   DATA[467,23] := 980.5178;
   DATA[467,24] := 2.0;
   DATA[467,25] := 2.0;
   DATA[467,26] := 7.878621;
   DATA[467,27] := 145.091;
   DATA[467,28] := 263.5222;
   DATA[467,29] := 12.11228;
   DATA[467,30] := 1.729557;
   DATA[467,31] := 1.292046;
   DATA[467,32] := 0.7353967;
   DATA[467,33] := 0.3065048;
   DATA[467,34] := 2.0;
   DATA[467,35] := 251.2817;
   DATA[467,36] := 1.746067;
   DATA[467,37] := 190.0634;
   DATA[467,38] := 0.000128152;
   DATA[467,39] := 1.0;
   DATA[468,0] := 2.44243;
   DATA[468,1] := 530.9328;
   DATA[468,2] := 2.0;
   DATA[468,3] := 2.0;
   DATA[468,4] := 262.1764;
   DATA[468,5] := 8.394835;
   DATA[468,6] := 327.9928;
   DATA[468,7] := 2.440521;
   DATA[468,8] := 2.0;
   DATA[468,9] := 2.0;
   DATA[468,10] := 2.0;
   DATA[468,11] := 19.69396;
   DATA[468,12] := 2.213881;
   DATA[468,13] := 980.0773;
   DATA[468,14] := 1.0;
   DATA[468,15] := 2.0;
   DATA[468,16] := 1.0;
   DATA[468,17] := 1.0;
   DATA[468,18] := 1.0;
   DATA[468,19] := 2.0;
   DATA[468,20] := 148.808;
   DATA[468,21] := 155.96;
   DATA[468,22] := 1.720565;
   DATA[468,23] := 980.5563;
   DATA[468,24] := 2.0;
   DATA[468,25] := 2.0;
   DATA[468,26] := 7.878621;
   DATA[468,27] := 145.091;
   DATA[468,28] := 263.5222;
   DATA[468,29] := 12.11228;
   DATA[468,30] := 1.730838;
   DATA[468,31] := 1.293198;
   DATA[468,32] := 0.7353967;
   DATA[468,33] := 0.3065048;
   DATA[468,34] := 2.0;
   DATA[468,35] := 251.2817;
   DATA[468,36] := 1.826162;
   DATA[468,37] := 190.0634;
   DATA[468,38] := 0.000128152;
   DATA[468,39] := 1.0;
   DATA[469,0] := 2.427377;
   DATA[469,1] := 530.3832;
   DATA[469,2] := 2.0;
   DATA[469,3] := 2.0;
   DATA[469,4] := 262.1764;
   DATA[469,5] := 8.394835;
   DATA[469,6] := 327.9928;
   DATA[469,7] := 2.440137;
   DATA[469,8] := 2.0;
   DATA[469,9] := 2.0;
   DATA[469,10] := 2.0;
   DATA[469,11] := 19.69396;
   DATA[469,12] := 2.213881;
   DATA[469,13] := 979.9971;
   DATA[469,14] := 1.0;
   DATA[469,15] := 2.0;
   DATA[469,16] := 1.0;
   DATA[469,17] := 1.0;
   DATA[469,18] := 1.0;
   DATA[469,19] := 2.0;
   DATA[469,20] := 148.808;
   DATA[469,21] := 155.96;
   DATA[469,22] := 1.720565;
   DATA[469,23] := 980.5563;
   DATA[469,24] := 2.0;
   DATA[469,25] := 2.0;
   DATA[469,26] := 7.878621;
   DATA[469,27] := 145.091;
   DATA[469,28] := 263.5222;
   DATA[469,29] := 12.11228;
   DATA[469,30] := 1.730838;
   DATA[469,31] := 1.296657;
   DATA[469,32] := 0.7353967;
   DATA[469,33] := 0.3065048;
   DATA[469,34] := 2.0;
   DATA[469,35] := 251.2817;
   DATA[469,36] := 1.826162;
   DATA[469,37] := 190.0634;
   DATA[469,38] := 0.000128152;
   DATA[469,39] := 1.0;
   DATA[470,0] := 2.427377;
   DATA[470,1] := 530.6188;
   DATA[470,2] := 2.0;
   DATA[470,3] := 2.0;
   DATA[470,4] := 262.1764;
   DATA[470,5] := 8.394835;
   DATA[470,6] := 327.9928;
   DATA[470,7] := 2.440137;
   DATA[470,8] := 2.0;
   DATA[470,9] := 2.0;
   DATA[470,10] := 2.0;
   DATA[470,11] := 19.65235;
   DATA[470,12] := 2.213881;
   DATA[470,13] := 979.9571;
   DATA[470,14] := 1.0;
   DATA[470,15] := 2.0;
   DATA[470,16] := 1.0;
   DATA[470,17] := 1.0;
   DATA[470,18] := 1.0;
   DATA[470,19] := 2.0;
   DATA[470,20] := 148.808;
   DATA[470,21] := 155.96;
   DATA[470,22] := 1.720565;
   DATA[470,23] := 980.364;
   DATA[470,24] := 2.0;
   DATA[470,25] := 2.0;
   DATA[470,26] := 7.878621;
   DATA[470,27] := 145.091;
   DATA[470,28] := 263.5222;
   DATA[470,29] := 12.11228;
   DATA[470,30] := 1.730838;
   DATA[470,31] := 1.289868;
   DATA[470,32] := 0.7353967;
   DATA[470,33] := 0.3065048;
   DATA[470,34] := 2.0;
   DATA[470,35] := 251.2817;
   DATA[470,36] := 1.762086;
   DATA[470,37] := 190.0634;
   DATA[470,38] := 0.000128152;
   DATA[470,39] := 1.0;
   DATA[471,0] := 2.427377;
   DATA[471,1] := 530.3047;
   DATA[471,2] := 2.0;
   DATA[471,3] := 2.0;
   DATA[471,4] := 262.1764;
   DATA[471,5] := 8.394835;
   DATA[471,6] := 327.9928;
   DATA[471,7] := 2.440137;
   DATA[471,8] := 2.0;
   DATA[471,9] := 2.0;
   DATA[471,10] := 2.0;
   DATA[471,11] := 19.65235;
   DATA[471,12] := 2.213881;
   DATA[471,13] := 980.1573;
   DATA[471,14] := 1.0;
   DATA[471,15] := 2.0;
   DATA[471,16] := 1.0;
   DATA[471,17] := 1.0;
   DATA[471,18] := 1.0;
   DATA[471,19] := 2.0;
   DATA[471,20] := 148.808;
   DATA[471,21] := 155.96;
   DATA[471,22] := 1.720565;
   DATA[471,23] := 980.7101;
   DATA[471,24] := 2.0;
   DATA[471,25] := 2.0;
   DATA[471,26] := 7.878621;
   DATA[471,27] := 145.091;
   DATA[471,28] := 263.5222;
   DATA[471,29] := 12.11228;
   DATA[471,30] := 1.730838;
   DATA[471,31] := 1.289868;
   DATA[471,32] := 0.7352687;
   DATA[471,33] := 0.3065048;
   DATA[471,34] := 2.0;
   DATA[471,35] := 251.2817;
   DATA[471,36] := 1.69801;
   DATA[471,37] := 190.0634;
   DATA[471,38] := 0.000128152;
   DATA[471,39] := 1.0;
   DATA[472,0] := 2.447234;
   DATA[472,1] := 530.6973;
   DATA[472,2] := 2.0;
   DATA[472,3] := 2.0;
   DATA[472,4] := 262.1764;
   DATA[472,5] := 8.394835;
   DATA[472,6] := 327.9928;
   DATA[472,7] := 2.440137;
   DATA[472,8] := 2.0;
   DATA[472,9] := 2.0;
   DATA[472,10] := 2.0;
   DATA[472,11] := 19.65235;
   DATA[472,12] := 2.213881;
   DATA[472,13] := 980.2775;
   DATA[472,14] := 1.0;
   DATA[472,15] := 2.0;
   DATA[472,16] := 1.0;
   DATA[472,17] := 1.0;
   DATA[472,18] := 1.0;
   DATA[472,19] := 2.0;
   DATA[472,20] := 148.808;
   DATA[472,21] := 155.96;
   DATA[472,22] := 1.720565;
   DATA[472,23] := 980.5178;
   DATA[472,24] := 2.0;
   DATA[472,25] := 2.0;
   DATA[472,26] := 7.878621;
   DATA[472,27] := 145.091;
   DATA[472,28] := 263.5222;
   DATA[472,29] := 12.11228;
   DATA[472,30] := 1.730838;
   DATA[472,31] := 1.288331;
   DATA[472,32] := 0.7352687;
   DATA[472,33] := 0.3065048;
   DATA[472,34] := 2.0;
   DATA[472,35] := 251.2817;
   DATA[472,36] := 1.69801;
   DATA[472,37] := 190.0634;
   DATA[472,38] := 0.000128152;
   DATA[472,39] := 1.0;
   DATA[473,0] := 2.496237;
   DATA[473,1] := 531.0898;
   DATA[473,2] := 2.0;
   DATA[473,3] := 2.0;
   DATA[473,4] := 262.1764;
   DATA[473,5] := 8.394835;
   DATA[473,6] := 327.9928;
   DATA[473,7] := 2.440137;
   DATA[473,8] := 2.0;
   DATA[473,9] := 2.0;
   DATA[473,10] := 2.0;
   DATA[473,11] := 19.65235;
   DATA[473,12] := 2.2126;
   DATA[473,13] := 980.5579;
   DATA[473,14] := 1.0;
   DATA[473,15] := 2.0;
   DATA[473,16] := 1.0;
   DATA[473,17] := 1.0;
   DATA[473,18] := 1.0;
   DATA[473,19] := 2.0;
   DATA[473,20] := 148.808;
   DATA[473,21] := 155.96;
   DATA[473,22] := 1.720565;
   DATA[473,23] := 980.4409;
   DATA[473,24] := 2.0;
   DATA[473,25] := 2.0;
   DATA[473,26] := 7.878621;
   DATA[473,27] := 145.091;
   DATA[473,28] := 263.4901;
   DATA[473,29] := 12.11228;
   DATA[473,30] := 1.730838;
   DATA[473,31] := 1.285641;
   DATA[473,32] := 0.7352687;
   DATA[473,33] := 0.3065048;
   DATA[473,34] := 2.0;
   DATA[473,35] := 251.2817;
   DATA[473,36] := 1.69801;
   DATA[473,37] := 190.0634;
   DATA[473,38] := 0.000128152;
   DATA[473,39] := 1.0;
   DATA[474,0] := 2.532108;
   DATA[474,1] := 531.5609;
   DATA[474,2] := 2.0;
   DATA[474,3] := 2.0;
   DATA[474,4] := 262.1764;
   DATA[474,5] := 8.394835;
   DATA[474,6] := 327.9928;
   DATA[474,7] := 2.440137;
   DATA[474,8] := 2.0;
   DATA[474,9] := 2.0;
   DATA[474,10] := 2.0;
   DATA[474,11] := 19.65235;
   DATA[474,12] := 2.2126;
   DATA[474,13] := 980.4377;
   DATA[474,14] := 1.0;
   DATA[474,15] := 2.0;
   DATA[474,16] := 1.0;
   DATA[474,17] := 1.0;
   DATA[474,18] := 1.0;
   DATA[474,19] := 2.0;
   DATA[474,20] := 148.808;
   DATA[474,21] := 155.96;
   DATA[474,22] := 1.720565;
   DATA[474,23] := 980.5563;
   DATA[474,24] := 2.0;
   DATA[474,25] := 2.0;
   DATA[474,26] := 7.878621;
   DATA[474,27] := 145.091;
   DATA[474,28] := 263.4901;
   DATA[474,29] := 12.11228;
   DATA[474,30] := 1.730838;
   DATA[474,31] := 1.301652;
   DATA[474,32] := 0.7352687;
   DATA[474,33] := 0.3066329;
   DATA[474,34] := 2.0;
   DATA[474,35] := 251.2817;
   DATA[474,36] := 1.69801;
   DATA[474,37] := 190.0634;
   DATA[474,38] := 0.000128152;
   DATA[474,39] := 1.0;
   DATA[475,0] := 2.577267;
   DATA[475,1] := 531.6786;
   DATA[475,2] := 2.0;
   DATA[475,3] := 2.0;
   DATA[475,4] := 262.1764;
   DATA[475,5] := 8.394835;
   DATA[475,6] := 327.9928;
   DATA[475,7] := 2.440137;
   DATA[475,8] := 2.0;
   DATA[475,9] := 2.0;
   DATA[475,10] := 2.0;
   DATA[475,11] := 19.65235;
   DATA[475,12] := 2.2126;
   DATA[475,13] := 980.3576;
   DATA[475,14] := 1.0;
   DATA[475,15] := 2.0;
   DATA[475,16] := 1.0;
   DATA[475,17] := 1.0;
   DATA[475,18] := 1.0;
   DATA[475,19] := 2.0;
   DATA[475,20] := 148.808;
   DATA[475,21] := 155.96;
   DATA[475,22] := 1.720565;
   DATA[475,23] := 980.7485;
   DATA[475,24] := 2.0;
   DATA[475,25] := 2.0;
   DATA[475,26] := 7.878621;
   DATA[475,27] := 145.091;
   DATA[475,28] := 263.4901;
   DATA[475,29] := 12.11228;
   DATA[475,30] := 1.730838;
   DATA[475,31] := 1.311387;
   DATA[475,32] := 0.7352687;
   DATA[475,33] := 0.3066329;
   DATA[475,34] := 2.0;
   DATA[475,35] := 251.2817;
   DATA[475,36] := 1.69801;
   DATA[475,37] := 190.0634;
   DATA[475,38] := 0.000128152;
   DATA[475,39] := 1.0;
   DATA[476,0] := 2.607373;
   DATA[476,1] := 532.1104;
   DATA[476,2] := 2.0;
   DATA[476,3] := 2.0;
   DATA[476,4] := 262.1764;
   DATA[476,5] := 8.394835;
   DATA[476,6] := 327.9928;
   DATA[476,7] := 2.440137;
   DATA[476,8] := 2.0;
   DATA[476,9] := 2.0;
   DATA[476,10] := 2.0;
   DATA[476,11] := 19.62033;
   DATA[476,12] := 2.2126;
   DATA[476,13] := 980.1573;
   DATA[476,14] := 1.0;
   DATA[476,15] := 2.0;
   DATA[476,16] := 1.0;
   DATA[476,17] := 1.0;
   DATA[476,18] := 1.0;
   DATA[476,19] := 2.0;
   DATA[476,20] := 148.808;
   DATA[476,21] := 155.96;
   DATA[476,22] := 1.722359;
   DATA[476,23] := 980.8254;
   DATA[476,24] := 2.0;
   DATA[476,25] := 2.0;
   DATA[476,26] := 7.878621;
   DATA[476,27] := 145.091;
   DATA[476,28] := 263.4901;
   DATA[476,29] := 12.11228;
   DATA[476,30] := 1.730838;
   DATA[476,31] := 1.32125;
   DATA[476,32] := 0.7352687;
   DATA[476,33] := 0.3066329;
   DATA[476,34] := 2.0;
   DATA[476,35] := 251.2817;
   DATA[476,36] := 1.69801;
   DATA[476,37] := 190.0634;
   DATA[476,38] := 0.000128152;
   DATA[476,39] := 1.0;
   DATA[477,0] := 2.637158;
   DATA[477,1] := 531.9141;
   DATA[477,2] := 2.0;
   DATA[477,3] := 2.0;
   DATA[477,4] := 262.1764;
   DATA[477,5] := 8.394835;
   DATA[477,6] := 327.9928;
   DATA[477,7] := 2.440137;
   DATA[477,8] := 2.0;
   DATA[477,9] := 2.0;
   DATA[477,10] := 2.0;
   DATA[477,11] := 19.69076;
   DATA[477,12] := 2.2126;
   DATA[477,13] := 979.9971;
   DATA[477,14] := 1.0;
   DATA[477,15] := 2.0;
   DATA[477,16] := 1.0;
   DATA[477,17] := 1.0;
   DATA[477,18] := 1.0;
   DATA[477,19] := 2.0;
   DATA[477,20] := 148.808;
   DATA[477,21] := 155.8575;
   DATA[477,22] := 1.724153;
   DATA[477,23] := 980.4409;
   DATA[477,24] := 2.0;
   DATA[477,25] := 2.0;
   DATA[477,26] := 7.878621;
   DATA[477,27] := 145.091;
   DATA[477,28] := 263.4901;
   DATA[477,29] := 12.11228;
   DATA[477,30] := 1.731479;
   DATA[477,31] := 1.320225;
   DATA[477,32] := 0.7352687;
   DATA[477,33] := 0.3066329;
   DATA[477,34] := 2.0;
   DATA[477,35] := 251.3939;
   DATA[477,36] := 1.69801;
   DATA[477,37] := 190.0634;
   DATA[477,38] := 0.000128152;
   DATA[477,39] := 1.0;
   DATA[478,0] := 2.649649;
   DATA[478,1] := 531.4824;
   DATA[478,2] := 2.0;
   DATA[478,3] := 2.0;
   DATA[478,4] := 262.1764;
   DATA[478,5] := 8.391951;
   DATA[478,6] := 327.9928;
   DATA[478,7] := 2.44206;
   DATA[478,8] := 2.0;
   DATA[478,9] := 2.0;
   DATA[478,10] := 2.0;
   DATA[478,11] := 19.71957;
   DATA[478,12] := 2.2126;
   DATA[478,13] := 979.9571;
   DATA[478,14] := 1.0;
   DATA[478,15] := 2.0;
   DATA[478,16] := 1.0;
   DATA[478,17] := 1.0;
   DATA[478,18] := 1.0;
   DATA[478,19] := 2.0;
   DATA[478,20] := 148.808;
   DATA[478,21] := 155.8575;
   DATA[478,22] := 1.724153;
   DATA[478,23] := 980.7485;
   DATA[478,24] := 2.0;
   DATA[478,25] := 2.0;
   DATA[478,26] := 7.878621;
   DATA[478,27] := 145.091;
   DATA[478,28] := 263.4901;
   DATA[478,29] := 12.11228;
   DATA[478,30] := 1.731479;
   DATA[478,31] := 1.312284;
   DATA[478,32] := 0.7352687;
   DATA[478,33] := 0.3066329;
   DATA[478,34] := 2.0;
   DATA[478,35] := 251.3939;
   DATA[478,36] := 1.69801;
   DATA[478,37] := 190.0634;
   DATA[478,38] := 0.000128152;
   DATA[478,39] := 1.0;
   DATA[479,0] := 2.652211;
   DATA[479,1] := 531.0898;
   DATA[479,2] := 2.0;
   DATA[479,3] := 2.0;
   DATA[479,4] := 262.1764;
   DATA[479,5] := 8.390669;
   DATA[479,6] := 327.9928;
   DATA[479,7] := 2.442188;
   DATA[479,8] := 2.0;
   DATA[479,9] := 2.0;
   DATA[479,10] := 2.0;
   DATA[479,11] := 19.76439;
   DATA[479,12] := 2.2126;
   DATA[479,13] := 980.1974;
   DATA[479,14] := 1.0;
   DATA[479,15] := 2.0;
   DATA[479,16] := 1.0;
   DATA[479,17] := 1.0;
   DATA[479,18] := 1.0;
   DATA[479,19] := 2.0;
   DATA[479,20] := 148.808;
   DATA[479,21] := 155.8575;
   DATA[479,22] := 1.722872;
   DATA[479,23] := 981.1331;
   DATA[479,24] := 2.0;
   DATA[479,25] := 2.0;
   DATA[479,26] := 7.878621;
   DATA[479,27] := 145.091;
   DATA[479,28] := 263.4901;
   DATA[479,29] := 12.11228;
   DATA[479,30] := 1.731479;
   DATA[479,31] := 1.295376;
   DATA[479,32] := 0.7352687;
   DATA[479,33] := 0.3066329;
   DATA[479,34] := 2.0;
   DATA[479,35] := 251.3939;
   DATA[479,36] := 1.69801;
   DATA[479,37] := 190.0634;
   DATA[479,38] := 0.000128152;
   DATA[479,39] := 1.0;
   DATA[480,0] := 2.642923;
   DATA[480,1] := 530.4225;
   DATA[480,2] := 2.0;
   DATA[480,3] := 2.0;
   DATA[480,4] := 262.1764;
   DATA[480,5] := 8.390669;
   DATA[480,6] := 327.9928;
   DATA[480,7] := 2.442188;
   DATA[480,8] := 2.0;
   DATA[480,9] := 2.0;
   DATA[480,10] := 2.0;
   DATA[480,11] := 19.77399;
   DATA[480,12] := 2.2126;
   DATA[480,13] := 979.7568;
   DATA[480,14] := 1.0;
   DATA[480,15] := 2.0;
   DATA[480,16] := 1.0;
   DATA[480,17] := 1.0;
   DATA[480,18] := 1.0;
   DATA[480,19] := 2.0;
   DATA[480,20] := 148.808;
   DATA[480,21] := 155.8575;
   DATA[480,22] := 1.721847;
   DATA[480,23] := 980.8254;
   DATA[480,24] := 2.0;
   DATA[480,25] := 2.0;
   DATA[480,26] := 7.879582;
   DATA[480,27] := 145.091;
   DATA[480,28] := 263.4901;
   DATA[480,29] := 12.11228;
   DATA[480,30] := 1.731479;
   DATA[480,31] := 1.291533;
   DATA[480,32] := 0.7352687;
   DATA[480,33] := 0.3066329;
   DATA[480,34] := 2.0;
   DATA[480,35] := 251.3939;
   DATA[480,36] := 1.69801;
   DATA[480,37] := 190.0634;
   DATA[480,38] := 0.000128152;
   DATA[480,39] := 1.0;
   DATA[481,0] := 2.624347;
   DATA[481,1] := 529.9515;
   DATA[481,2] := 2.0;
   DATA[481,3] := 2.0;
   DATA[481,4] := 262.1764;
   DATA[481,5] := 8.390669;
   DATA[481,6] := 327.9928;
   DATA[481,7] := 2.441419;
   DATA[481,8] := 2.0;
   DATA[481,9] := 2.0;
   DATA[481,10] := 2.0;
   DATA[481,11] := 19.70357;
   DATA[481,12] := 2.2126;
   DATA[481,13] := 979.4364;
   DATA[481,14] := 1.0;
   DATA[481,15] := 2.0;
   DATA[481,16] := 1.0;
   DATA[481,17] := 1.0;
   DATA[481,18] := 1.0;
   DATA[481,19] := 2.0;
   DATA[481,20] := 148.808;
   DATA[481,21] := 155.8575;
   DATA[481,22] := 1.721334;
   DATA[481,23] := 980.8254;
   DATA[481,24] := 2.0;
   DATA[481,25] := 2.0;
   DATA[481,26] := 7.880544;
   DATA[481,27] := 145.091;
   DATA[481,28] := 263.4901;
   DATA[481,29] := 12.11228;
   DATA[481,30] := 1.731479;
   DATA[481,31] := 1.297938;
   DATA[481,32] := 0.7352687;
   DATA[481,33] := 0.3066329;
   DATA[481,34] := 2.0;
   DATA[481,35] := 251.2176;
   DATA[481,36] := 1.69801;
   DATA[481,37] := 190.0634;
   DATA[481,38] := 0.000128152;
   DATA[481,39] := 1.0;
   DATA[482,0] := 2.621785;
   DATA[482,1] := 529.2057;
   DATA[482,2] := 2.0;
   DATA[482,3] := 2.0;
   DATA[482,4] := 262.1764;
   DATA[482,5] := 8.390669;
   DATA[482,6] := 327.9928;
   DATA[482,7] := 2.440521;
   DATA[482,8] := 2.0;
   DATA[482,9] := 2.0;
   DATA[482,10] := 2.0;
   DATA[482,11] := 19.70357;
   DATA[482,12] := 2.2126;
   DATA[482,13] := 979.4764;
   DATA[482,14] := 1.0;
   DATA[482,15] := 2.0;
   DATA[482,16] := 1.0;
   DATA[482,17] := 1.0;
   DATA[482,18] := 1.0;
   DATA[482,19] := 2.0;
   DATA[482,20] := 148.808;
   DATA[482,21] := 155.8575;
   DATA[482,22] := 1.720565;
   DATA[482,23] := 980.9023;
   DATA[482,24] := 2.0;
   DATA[482,25] := 2.0;
   DATA[482,26] := 7.880544;
   DATA[482,27] := 145.091;
   DATA[482,28] := 263.4901;
   DATA[482,29] := 12.11228;
   DATA[482,30] := 1.731479;
   DATA[482,31] := 1.302293;
   DATA[482,32] := 0.7352687;
   DATA[482,33] := 0.3066329;
   DATA[482,34] := 2.0;
   DATA[482,35] := 251.0734;
   DATA[482,36] := 1.69801;
   DATA[482,37] := 189.8872;
   DATA[482,38] := 0.000128152;
   DATA[482,39] := 1.0;
   DATA[483,0] := 2.613778;
   DATA[483,1] := 528.8132;
   DATA[483,2] := 2.0;
   DATA[483,3] := 2.0;
   DATA[483,4] := 262.1764;
   DATA[483,5] := 8.39131;
   DATA[483,6] := 327.9928;
   DATA[483,7] := 2.442828;
   DATA[483,8] := 2.0;
   DATA[483,9] := 2.0;
   DATA[483,10] := 2.0;
   DATA[483,11] := 19.70357;
   DATA[483,12] := 2.208628;
   DATA[483,13] := 979.5565;
   DATA[483,14] := 1.0;
   DATA[483,15] := 2.0;
   DATA[483,16] := 1.0;
   DATA[483,17] := 1.0;
   DATA[483,18] := 1.0;
   DATA[483,19] := 2.0;
   DATA[483,20] := 148.808;
   DATA[483,21] := 155.8575;
   DATA[483,22] := 1.720309;
   DATA[483,23] := 981.1331;
   DATA[483,24] := 2.0;
   DATA[483,25] := 2.0;
   DATA[483,26] := 7.880544;
   DATA[483,27] := 145.091;
   DATA[483,28] := 263.4901;
   DATA[483,29] := 12.11228;
   DATA[483,30] := 1.731479;
   DATA[483,31] := 1.310106;
   DATA[483,32] := 0.7352687;
   DATA[483,33] := 0.3066329;
   DATA[483,34] := 2.0;
   DATA[483,35] := 251.0734;
   DATA[483,36] := 1.69801;
   DATA[483,37] := 189.8872;
   DATA[483,38] := 0.000128152;
   DATA[483,39] := 1.0;
   DATA[484,0] := 2.60449;
   DATA[484,1] := 528.6169;
   DATA[484,2] := 2.0;
   DATA[484,3] := 2.0;
   DATA[484,4] := 262.1764;
   DATA[484,5] := 8.393553;
   DATA[484,6] := 327.9928;
   DATA[484,7] := 2.442828;
   DATA[484,8] := 2.0;
   DATA[484,9] := 2.0;
   DATA[484,10] := 2.0;
   DATA[484,11] := 19.65235;
   DATA[484,12] := 2.208628;
   DATA[484,13] := 979.0759;
   DATA[484,14] := 1.0;
   DATA[484,15] := 2.0;
   DATA[484,16] := 1.0;
   DATA[484,17] := 1.0;
   DATA[484,18] := 1.0;
   DATA[484,19] := 2.0;
   DATA[484,20] := 148.808;
   DATA[484,21] := 155.8575;
   DATA[484,22] := 1.720309;
   DATA[484,23] := 981.0946;
   DATA[484,24] := 2.0;
   DATA[484,25] := 2.0;
   DATA[484,26] := 7.880544;
   DATA[484,27] := 145.091;
   DATA[484,28] := 263.4901;
   DATA[484,29] := 12.11228;
   DATA[484,30] := 1.731479;
   DATA[484,31] := 1.312412;
   DATA[484,32] := 0.7352687;
   DATA[484,33] := 0.3066329;
   DATA[484,34] := 2.0;
   DATA[484,35] := 251.0734;
   DATA[484,36] := 1.69801;
   DATA[484,37] := 189.8872;
   DATA[484,38] := 0.000128152;
   DATA[484,39] := 1.0;
   DATA[485,0] := 2.587195;
   DATA[485,1] := 528.9309;
   DATA[485,2] := 2.0;
   DATA[485,3] := 2.0;
   DATA[485,4] := 262.1764;
   DATA[485,5] := 8.393553;
   DATA[485,6] := 327.9928;
   DATA[485,7] := 2.442828;
   DATA[485,8] := 2.0;
   DATA[485,9] := 2.0;
   DATA[485,10] := 2.0;
   DATA[485,11] := 19.65235;
   DATA[485,12] := 2.208628;
   DATA[485,13] := 979.2762;
   DATA[485,14] := 1.0;
   DATA[485,15] := 2.0;
   DATA[485,16] := 1.0;
   DATA[485,17] := 1.0;
   DATA[485,18] := 1.0;
   DATA[485,19] := 2.0;
   DATA[485,20] := 148.808;
   DATA[485,21] := 155.5755;
   DATA[485,22] := 1.719412;
   DATA[485,23] := 981.556;
   DATA[485,24] := 2.0;
   DATA[485,25] := 2.0;
   DATA[485,26] := 7.880544;
   DATA[485,27] := 145.091;
   DATA[485,28] := 263.4901;
   DATA[485,29] := 12.11228;
   DATA[485,30] := 1.731479;
   DATA[485,31] := 1.306264;
   DATA[485,32] := 0.7378293;
   DATA[485,33] := 0.3066329;
   DATA[485,34] := 2.0;
   DATA[485,35] := 251.0734;
   DATA[485,36] := 1.69801;
   DATA[485,37] := 189.8071;
   DATA[485,38] := 0.000128152;
   DATA[485,39] := 1.0;
   DATA[486,0] := 2.570541;
   DATA[486,1] := 528.9702;
   DATA[486,2] := 2.0;
   DATA[486,3] := 2.0;
   DATA[486,4] := 262.1764;
   DATA[486,5] := 8.393553;
   DATA[486,6] := 327.9928;
   DATA[486,7] := 2.441547;
   DATA[486,8] := 2.0;
   DATA[486,9] := 2.0;
   DATA[486,10] := 2.0;
   DATA[486,11] := 19.65235;
   DATA[486,12] := 2.209653;
   DATA[486,13] := 979.5966;
   DATA[486,14] := 1.0;
   DATA[486,15] := 2.0;
   DATA[486,16] := 1.0;
   DATA[486,17] := 1.0;
   DATA[486,18] := 1.0;
   DATA[486,19] := 2.0;
   DATA[486,20] := 148.808;
   DATA[486,21] := 155.5755;
   DATA[486,22] := 1.718771;
   DATA[486,23] := 981.4022;
   DATA[486,24] := 2.0;
   DATA[486,25] := 2.0;
   DATA[486,26] := 7.880544;
   DATA[486,27] := 145.091;
   DATA[486,28] := 263.4901;
   DATA[486,29] := 12.11228;
   DATA[486,30] := 1.731479;
   DATA[486,31] := 1.286153;
   DATA[486,32] := 0.7379573;
   DATA[486,33] := 0.3066329;
   DATA[486,34] := 2.0;
   DATA[486,35] := 251.0734;
   DATA[486,36] := 1.69801;
   DATA[486,37] := 189.6789;
   DATA[486,38] := 0.000128152;
   DATA[486,39] := 1.0;
   DATA[487,0] := 2.551324;
   DATA[487,1] := 529.402;
   DATA[487,2] := 2.0;
   DATA[487,3] := 2.0;
   DATA[487,4] := 262.1764;
   DATA[487,5] := 8.393553;
   DATA[487,6] := 327.9928;
   DATA[487,7] := 2.441547;
   DATA[487,8] := 2.0;
   DATA[487,9] := 2.0;
   DATA[487,10] := 2.0;
   DATA[487,11] := 19.65235;
   DATA[487,12] := 2.209909;
   DATA[487,13] := 979.156;
   DATA[487,14] := 1.0;
   DATA[487,15] := 2.0;
   DATA[487,16] := 1.0;
   DATA[487,17] := 1.0;
   DATA[487,18] := 1.0;
   DATA[487,19] := 2.0;
   DATA[487,20] := 148.808;
   DATA[487,21] := 155.5755;
   DATA[487,22] := 1.718771;
   DATA[487,23] := 981.4791;
   DATA[487,24] := 2.0;
   DATA[487,25] := 2.0;
   DATA[487,26] := 7.880544;
   DATA[487,27] := 145.091;
   DATA[487,28] := 263.4901;
   DATA[487,29] := 12.11228;
   DATA[487,30] := 1.731479;
   DATA[487,31] := 1.281798;
   DATA[487,32] := 0.7379573;
   DATA[487,33] := 0.3066329;
   DATA[487,34] := 2.0;
   DATA[487,35] := 251.0734;
   DATA[487,36] := 1.69801;
   DATA[487,37] := 189.6789;
   DATA[487,38] := 0.000128152;
   DATA[487,39] := 1.0;
   DATA[488,0] := 2.537552;
   DATA[488,1] := 529.7945;
   DATA[488,2] := 2.0;
   DATA[488,3] := 2.0;
   DATA[488,4] := 262.1764;
   DATA[488,5] := 8.393553;
   DATA[488,6] := 327.9928;
   DATA[488,7] := 2.439496;
   DATA[488,8] := 2.0;
   DATA[488,9] := 2.0;
   DATA[488,10] := 2.0;
   DATA[488,11] := 19.65235;
   DATA[488,12] := 2.209909;
   DATA[488,13] := 978.9958;
   DATA[488,14] := 1.0;
   DATA[488,15] := 2.0;
   DATA[488,16] := 1.0;
   DATA[488,17] := 1.0;
   DATA[488,18] := 1.0;
   DATA[488,19] := 2.0;
   DATA[488,20] := 148.808;
   DATA[488,21] := 155.5755;
   DATA[488,22] := 1.718771;
   DATA[488,23] := 981.7867;
   DATA[488,24] := 2.0;
   DATA[488,25] := 2.0;
   DATA[488,26] := 7.880544;
   DATA[488,27] := 145.091;
   DATA[488,28] := 263.4901;
   DATA[488,29] := 12.11228;
   DATA[488,30] := 1.731479;
   DATA[488,31] := 1.281798;
   DATA[488,32] := 0.7379573;
   DATA[488,33] := 0.3066329;
   DATA[488,34] := 2.0;
   DATA[488,35] := 251.0734;
   DATA[488,36] := 1.69801;
   DATA[488,37] := 189.6789;
   DATA[488,38] := 0.000128152;
   DATA[488,39] := 1.0;
   DATA[489,0] := 2.519937;
   DATA[489,1] := 530.3047;
   DATA[489,2] := 2.0;
   DATA[489,3] := 2.0;
   DATA[489,4] := 262.1764;
   DATA[489,5] := 8.393553;
   DATA[489,6] := 327.9928;
   DATA[489,7] := 2.439496;
   DATA[489,8] := 2.0;
   DATA[489,9] := 2.0;
   DATA[489,10] := 2.0;
   DATA[489,11] := 19.65235;
   DATA[489,12] := 2.209909;
   DATA[489,13] := 978.6353;
   DATA[489,14] := 1.0;
   DATA[489,15] := 2.0;
   DATA[489,16] := 1.0;
   DATA[489,17] := 1.0;
   DATA[489,18] := 1.0;
   DATA[489,19] := 2.0;
   DATA[489,20] := 148.808;
   DATA[489,21] := 155.5755;
   DATA[489,22] := 1.718771;
   DATA[489,23] := 981.7483;
   DATA[489,24] := 2.0;
   DATA[489,25] := 2.0;
   DATA[489,26] := 7.880544;
   DATA[489,27] := 145.091;
   DATA[489,28] := 263.4901;
   DATA[489,29] := 12.11228;
   DATA[489,30] := 1.731479;
   DATA[489,31] := 1.290124;
   DATA[489,32] := 0.7379573;
   DATA[489,33] := 0.3066329;
   DATA[489,34] := 2.0;
   DATA[489,35] := 251.0734;
   DATA[489,36] := 1.69801;
   DATA[489,37] := 189.8391;
   DATA[489,38] := 0.000128152;
   DATA[489,39] := 1.0;
   DATA[490,0] := 2.506485;
   DATA[490,1] := 530.7758;
   DATA[490,2] := 2.0;
   DATA[490,3] := 2.0;
   DATA[490,4] := 262.1764;
   DATA[490,5] := 8.393553;
   DATA[490,6] := 327.9928;
   DATA[490,7] := 2.440393;
   DATA[490,8] := 2.0;
   DATA[490,9] := 2.0;
   DATA[490,10] := 2.0;
   DATA[490,11] := 19.69076;
   DATA[490,12] := 2.209909;
   DATA[490,13] := 978.8356;
   DATA[490,14] := 1.0;
   DATA[490,15] := 2.0;
   DATA[490,16] := 1.0;
   DATA[490,17] := 1.0;
   DATA[490,18] := 1.0;
   DATA[490,19] := 2.0;
   DATA[490,20] := 148.808;
   DATA[490,21] := 155.5755;
   DATA[490,22] := 1.718771;
   DATA[490,23] := 981.9406;
   DATA[490,24] := 2.0;
   DATA[490,25] := 2.0;
   DATA[490,26] := 7.880544;
   DATA[490,27] := 145.091;
   DATA[490,28] := 263.4901;
   DATA[490,29] := 12.11228;
   DATA[490,30] := 1.729941;
   DATA[490,31] := 1.310106;
   DATA[490,32] := 0.7353967;
   DATA[490,33] := 0.3068891;
   DATA[490,34] := 2.0;
   DATA[490,35] := 251.0734;
   DATA[490,36] := 1.69801;
   DATA[490,37] := 189.8391;
   DATA[490,38] := 0.000128152;
   DATA[490,39] := 1.0;
   DATA[491,0] := 2.489831;
   DATA[491,1] := 531.2861;
   DATA[491,2] := 2.0;
   DATA[491,3] := 2.0;
   DATA[491,4] := 262.1764;
   DATA[491,5] := 8.393553;
   DATA[491,6] := 327.9928;
   DATA[491,7] := 2.440393;
   DATA[491,8] := 2.0;
   DATA[491,9] := 2.0;
   DATA[491,10] := 2.0;
   DATA[491,11] := 19.70997;
   DATA[491,12] := 2.209909;
   DATA[491,13] := 978.6353;
   DATA[491,14] := 1.0;
   DATA[491,15] := 2.0;
   DATA[491,16] := 1.0;
   DATA[491,17] := 1.0;
   DATA[491,18] := 1.0;
   DATA[491,19] := 2.0;
   DATA[491,20] := 148.808;
   DATA[491,21] := 155.7806;
   DATA[491,22] := 1.719027;
   DATA[491,23] := 982.1713;
   DATA[491,24] := 2.0;
   DATA[491,25] := 2.0;
   DATA[491,26] := 7.880544;
   DATA[491,27] := 145.091;
   DATA[491,28] := 263.4901;
   DATA[491,29] := 12.11228;
   DATA[491,30] := 1.728659;
   DATA[491,31] := 1.305367;
   DATA[491,32] := 0.7353967;
   DATA[491,33] := 0.3083624;
   DATA[491,34] := 2.0;
   DATA[491,35] := 251.0734;
   DATA[491,36] := 1.69801;
   DATA[491,37] := 189.8391;
   DATA[491,38] := 0.000128152;
   DATA[491,39] := 1.0;
   DATA[492,0] := 2.47638;
   DATA[492,1] := 531.6001;
   DATA[492,2] := 2.0;
   DATA[492,3] := 2.0;
   DATA[492,4] := 262.1764;
   DATA[492,5] := 8.393553;
   DATA[492,6] := 327.9928;
   DATA[492,7] := 2.440393;
   DATA[492,8] := 2.0;
   DATA[492,9] := 2.0;
   DATA[492,10] := 2.0;
   DATA[492,11] := 19.73238;
   DATA[492,12] := 2.209909;
   DATA[492,13] := 978.395;
   DATA[492,14] := 1.0;
   DATA[492,15] := 2.0;
   DATA[492,16] := 1.0;
   DATA[492,17] := 1.0;
   DATA[492,18] := 1.0;
   DATA[492,19] := 2.0;
   DATA[492,20] := 148.808;
   DATA[492,21] := 155.7806;
   DATA[492,22] := 1.720693;
   DATA[492,23] := 981.8636;
   DATA[492,24] := 2.0;
   DATA[492,25] := 2.0;
   DATA[492,26] := 7.880544;
   DATA[492,27] := 145.091;
   DATA[492,28] := 263.4901;
   DATA[492,29] := 12.11228;
   DATA[492,30] := 1.728659;
   DATA[492,31] := 1.301652;
   DATA[492,32] := 0.7353967;
   DATA[492,33] := 0.3083624;
   DATA[492,34] := 2.0;
   DATA[492,35] := 251.0734;
   DATA[492,36] := 1.69801;
   DATA[492,37] := 189.8391;
   DATA[492,38] := 0.000128152;
   DATA[492,39] := 1.0;
   DATA[493,0] := 2.458444;
   DATA[493,1] := 531.9534;
   DATA[493,2] := 2.0;
   DATA[493,3] := 2.0;
   DATA[493,4] := 262.1764;
   DATA[493,5] := 8.396437;
   DATA[493,6] := 327.9928;
   DATA[493,7] := 2.440393;
   DATA[493,8] := 2.0;
   DATA[493,9] := 2.0;
   DATA[493,10] := 2.0;
   DATA[493,11] := 19.73558;
   DATA[493,12] := 2.209909;
   DATA[493,13] := 978.2347;
   DATA[493,14] := 1.0;
   DATA[493,15] := 2.0;
   DATA[493,16] := 1.0;
   DATA[493,17] := 1.0;
   DATA[493,18] := 1.0;
   DATA[493,19] := 2.0;
   DATA[493,20] := 148.808;
   DATA[493,21] := 155.7806;
   DATA[493,22] := 1.720693;
   DATA[493,23] := 982.4404;
   DATA[493,24] := 2.0;
   DATA[493,25] := 2.0;
   DATA[493,26] := 7.880544;
   DATA[493,27] := 145.091;
   DATA[493,28] := 263.4901;
   DATA[493,29] := 12.11228;
   DATA[493,30] := 1.728659;
   DATA[493,31] := 1.292046;
   DATA[493,32] := 0.7353967;
   DATA[493,33] := 0.3083624;
   DATA[493,34] := 2.0;
   DATA[493,35] := 251.0734;
   DATA[493,36] := 1.69801;
   DATA[493,37] := 189.8391;
   DATA[493,38] := 0.000128152;
   DATA[493,39] := 1.0;
   DATA[494,0] := 2.440829;
   DATA[494,1] := 531.9926;
   DATA[494,2] := 2.0;
   DATA[494,3] := 2.0;
   DATA[494,4] := 262.1764;
   DATA[494,5] := 8.396437;
   DATA[494,6] := 327.9928;
   DATA[494,7] := 2.440393;
   DATA[494,8] := 2.0;
   DATA[494,9] := 2.0;
   DATA[494,10] := 2.0;
   DATA[494,11] := 19.73558;
   DATA[494,12] := 2.209909;
   DATA[494,13] := 978.1547;
   DATA[494,14] := 1.0;
   DATA[494,15] := 2.0;
   DATA[494,16] := 1.0;
   DATA[494,17] := 1.0;
   DATA[494,18] := 1.0;
   DATA[494,19] := 2.0;
   DATA[494,20] := 148.808;
   DATA[494,21] := 155.5499;
   DATA[494,22] := 1.720693;
   DATA[494,23] := 982.3251;
   DATA[494,24] := 2.0;
   DATA[494,25] := 2.0;
   DATA[494,26] := 7.880544;
   DATA[494,27] := 145.091;
   DATA[494,28] := 263.4901;
   DATA[494,29] := 12.11228;
   DATA[494,30] := 1.726737;
   DATA[494,31] := 1.291789;
   DATA[494,32] := 0.7353967;
   DATA[494,33] := 0.3083624;
   DATA[494,34] := 2.0;
   DATA[494,35] := 250.9773;
   DATA[494,36] := 1.69801;
   DATA[494,37] := 189.8391;
   DATA[494,38] := 0.000128152;
   DATA[494,39] := 1.0;
   DATA[495,0] := 2.440829;
   DATA[495,1] := 531.9926;
   DATA[495,2] := 2.0;
   DATA[495,3] := 2.0;
   DATA[495,4] := 262.1764;
   DATA[495,5] := 8.396437;
   DATA[495,6] := 327.9928;
   DATA[495,7] := 2.440393;
   DATA[495,8] := 2.0;
   DATA[495,9] := 2.0;
   DATA[495,10] := 2.0;
   DATA[495,11] := 19.73558;
   DATA[495,12] := 2.209909;
   DATA[495,13] := 978.1547;
   DATA[495,14] := 1.0;
   DATA[495,15] := 2.0;
   DATA[495,16] := 1.0;
   DATA[495,17] := 1.0;
   DATA[495,18] := 1.0;
   DATA[495,19] := 2.0;
   DATA[495,20] := 148.808;
   DATA[495,21] := 155.5499;
   DATA[495,22] := 1.720693;
   DATA[495,23] := 982.3251;
   DATA[495,24] := 2.0;
   DATA[495,25] := 2.0;
   DATA[495,26] := 7.880544;
   DATA[495,27] := 145.091;
   DATA[495,28] := 263.4901;
   DATA[495,29] := 12.11228;
   DATA[495,30] := 1.726737;
   DATA[495,31] := 1.291789;
   DATA[495,32] := 0.7353967;
   DATA[495,33] := 0.3083624;
   DATA[495,34] := 2.0;
   DATA[495,35] := 250.9773;
   DATA[495,36] := 1.69801;
   DATA[495,37] := 189.8391;
   DATA[495,38] := 0.000128152;
   DATA[495,39] := 1.0;
   DATA[496,0] := 2.43058;
   DATA[496,1] := 532.1104;
   DATA[496,2] := 2.0;
   DATA[496,3] := 2.0;
   DATA[496,4] := 262.1764;
   DATA[496,5] := 8.396437;
   DATA[496,6] := 327.9928;
   DATA[496,7] := 2.440393;
   DATA[496,8] := 2.0;
   DATA[496,9] := 2.0;
   DATA[496,10] := 2.0;
   DATA[496,11] := 19.73558;
   DATA[496,12] := 2.209909;
   DATA[496,13] := 978.2347;
   DATA[496,14] := 1.0;
   DATA[496,15] := 2.0;
   DATA[496,16] := 1.0;
   DATA[496,17] := 1.0;
   DATA[496,18] := 1.0;
   DATA[496,19] := 2.0;
   DATA[496,20] := 148.808;
   DATA[496,21] := 155.5499;
   DATA[496,22] := 1.720693;
   DATA[496,23] := 982.748;
   DATA[496,24] := 2.0;
   DATA[496,25] := 2.0;
   DATA[496,26] := 7.880544;
   DATA[496,27] := 145.091;
   DATA[496,28] := 263.4901;
   DATA[496,29] := 12.11228;
   DATA[496,30] := 1.726224;
   DATA[496,31] := 1.291789;
   DATA[496,32] := 0.7353967;
   DATA[496,33] := 0.3083624;
   DATA[496,34] := 2.0;
   DATA[496,35] := 250.9613;
   DATA[496,36] := 1.69801;
   DATA[496,37] := 189.759;
   DATA[496,38] := 0.000128152;
   DATA[496,39] := 1.0;
   DATA[497,0] := 2.424174;
   DATA[497,1] := 532.2674;
   DATA[497,2] := 2.0;
   DATA[497,3] := 2.0;
   DATA[497,4] := 262.1764;
   DATA[497,5] := 8.396437;
   DATA[497,6] := 328.0954;
   DATA[497,7] := 2.440393;
   DATA[497,8] := 2.0;
   DATA[497,9] := 2.0;
   DATA[497,10] := 2.0;
   DATA[497,11] := 19.73558;
   DATA[497,12] := 2.208372;
   DATA[497,13] := 978.2347;
   DATA[497,14] := 1.0;
   DATA[497,15] := 2.0;
   DATA[497,16] := 1.0;
   DATA[497,17] := 1.0;
   DATA[497,18] := 1.0;
   DATA[497,19] := 2.0;
   DATA[497,20] := 148.808;
   DATA[497,21] := 155.5499;
   DATA[497,22] := 1.720693;
   DATA[497,23] := 982.8249;
   DATA[497,24] := 2.0;
   DATA[497,25] := 2.0;
   DATA[497,26] := 7.880544;
   DATA[497,27] := 145.091;
   DATA[497,28] := 263.4901;
   DATA[497,29] := 12.11228;
   DATA[497,30] := 1.726224;
   DATA[497,31] := 1.299091;
   DATA[497,32] := 0.7353967;
   DATA[497,33] := 0.3083624;
   DATA[497,34] := 2.0;
   DATA[497,35] := 250.9613;
   DATA[497,36] := 1.69801;
   DATA[497,37] := 189.759;
   DATA[497,38] := 0.000128152;
   DATA[497,39] := 1.0;
   DATA[498,0] := 2.423534;
   DATA[498,1] := 532.4637;
   DATA[498,2] := 2.0;
   DATA[498,3] := 2.0;
   DATA[498,4] := 262.1764;
   DATA[498,5] := 8.396437;
   DATA[498,6] := 328.0954;
   DATA[498,7] := 2.440393;
   DATA[498,8] := 2.0;
   DATA[498,9] := 2.0;
   DATA[498,10] := 2.0;
   DATA[498,11] := 19.73558;
   DATA[498,12] := 2.206963;
   DATA[498,13] := 978.3549;
   DATA[498,14] := 1.0;
   DATA[498,15] := 2.0;
   DATA[498,16] := 1.0;
   DATA[498,17] := 1.0;
   DATA[498,18] := 1.0;
   DATA[498,19] := 2.0;
   DATA[498,20] := 148.808;
   DATA[498,21] := 155.7293;
   DATA[498,22] := 1.719284;
   DATA[498,23] := 983.2863;
   DATA[498,24] := 2.0;
   DATA[498,25] := 2.0;
   DATA[498,26] := 7.880544;
   DATA[498,27] := 145.091;
   DATA[498,28] := 263.4901;
   DATA[498,29] := 12.11228;
   DATA[498,30] := 1.728659;
   DATA[498,31] := 1.301396;
   DATA[498,32] := 0.7353967;
   DATA[498,33] := 0.3083624;
   DATA[498,34] := 2.0;
   DATA[498,35] := 250.9613;
   DATA[498,36] := 1.69801;
   DATA[498,37] := 189.759;
   DATA[498,38] := 0.000128152;
   DATA[498,39] := 1.0;
   DATA[499,0] := 2.452679;
   DATA[499,1] := 532.4637;
   DATA[499,2] := 2.0;
   DATA[499,3] := 2.0;
   DATA[499,4] := 262.1764;
   DATA[499,5] := 8.396437;
   DATA[499,6] := 328.0954;
   DATA[499,7] := 2.440393;
   DATA[499,8] := 2.0;
   DATA[499,9] := 2.0;
   DATA[499,10] := 2.0;
   DATA[499,11] := 19.73558;
   DATA[499,12] := 2.206963;
   DATA[499,13] := 978.4351;
   DATA[499,14] := 1.0;
   DATA[499,15] := 2.0;
   DATA[499,16] := 1.0;
   DATA[499,17] := 1.0;
   DATA[499,18] := 1.0;
   DATA[499,19] := 2.0;
   DATA[499,20] := 148.808;
   DATA[499,21] := 155.7293;
   DATA[499,22] := 1.719284;
   DATA[499,23] := 983.0941;
   DATA[499,24] := 2.0;
   DATA[499,25] := 2.0;
   DATA[499,26] := 7.880544;
   DATA[499,27] := 145.091;
   DATA[499,28] := 263.4901;
   DATA[499,29] := 12.11228;
   DATA[499,30] := 1.728659;
   DATA[499,31] := 1.292558;
   DATA[499,32] := 0.7353967;
   DATA[499,33] := 0.3069532;
   DATA[499,34] := 2.0;
   DATA[499,35] := 250.9613;
   DATA[499,36] := 1.730048;
   DATA[499,37] := 189.759;
   DATA[499,38] := 0.000128152;
   DATA[499,39] := 1.0;
   DATA[500,0] := 2.504884;
   DATA[500,1] := 532.3851;
   DATA[500,2] := 2.0;
   DATA[500,3] := 2.0;
   DATA[500,4] := 262.1764;
   DATA[500,5] := 8.396437;
   DATA[500,6] := 328.0954;
   DATA[500,7] := 2.440393;
   DATA[500,8] := 2.0;
   DATA[500,9] := 2.0;
   DATA[500,10] := 2.0;
   DATA[500,11] := 19.73558;
   DATA[500,12] := 2.206963;
   DATA[500,13] := 978.2748;
   DATA[500,14] := 1.0;
   DATA[500,15] := 2.0;
   DATA[500,16] := 1.0;
   DATA[500,17] := 1.0;
   DATA[500,18] := 1.0;
   DATA[500,19] := 2.0;
   DATA[500,20] := 148.808;
   DATA[500,21] := 155.7293;
   DATA[500,22] := 1.719284;
   DATA[500,23] := 983.1325;
   DATA[500,24] := 2.0;
   DATA[500,25] := 2.0;
   DATA[500,26] := 7.880544;
   DATA[500,27] := 145.091;
   DATA[500,28] := 263.4901;
   DATA[500,29] := 12.22763;
   DATA[500,30] := 1.729172;
   DATA[500,31] := 1.279365;
   DATA[500,32] := 0.7353967;
   DATA[500,33] := 0.3065048;
   DATA[500,34] := 2.0;
   DATA[500,35] := 250.9613;
   DATA[500,36] := 1.842181;
   DATA[500,37] := 189.759;
   DATA[500,38] := 0.000128152;
   DATA[500,39] := 1.0;
   DATA[501,0] := 2.545559;
   DATA[501,1] := 532.1104;
   DATA[501,2] := 2.0;
   DATA[501,3] := 2.0;
   DATA[501,4] := 262.1764;
   DATA[501,5] := 8.393873;
   DATA[501,6] := 328.0954;
   DATA[501,7] := 2.442316;
   DATA[501,8] := 2.0;
   DATA[501,9] := 2.0;
   DATA[501,10] := 2.0;
   DATA[501,11] := 19.73558;
   DATA[501,12] := 2.206963;
   DATA[501,13] := 978.0746;
   DATA[501,14] := 1.0;
   DATA[501,15] := 2.0;
   DATA[501,16] := 1.0;
   DATA[501,17] := 1.0;
   DATA[501,18] := 1.0;
   DATA[501,19] := 2.0;
   DATA[501,20] := 148.808;
   DATA[501,21] := 155.7293;
   DATA[501,22] := 1.719284;
   DATA[501,23] := 983.2863;
   DATA[501,24] := 2.0;
   DATA[501,25] := 2.0;
   DATA[501,26] := 7.880544;
   DATA[501,27] := 145.091;
   DATA[501,28] := 263.4901;
   DATA[501,29] := 12.22763;
   DATA[501,30] := 1.729172;
   DATA[501,31] := 1.262457;
   DATA[501,32] := 0.7353967;
   DATA[501,33] := 0.3065048;
   DATA[501,34] := 2.0;
   DATA[501,35] := 250.9613;
   DATA[501,36] := 1.842181;
   DATA[501,37] := 189.759;
   DATA[501,38] := 0.000128152;
   DATA[501,39] := 1.0;
   DATA[502,0] := 2.575345;
   DATA[502,1] := 532.3066;
   DATA[502,2] := 2.0;
   DATA[502,3] := 2.0;
   DATA[502,4] := 262.1764;
   DATA[502,5] := 8.393873;
   DATA[502,6] := 327.9159;
   DATA[502,7] := 2.443085;
   DATA[502,8] := 2.0;
   DATA[502,9] := 2.0;
   DATA[502,10] := 2.0;
   DATA[502,11] := 19.73558;
   DATA[502,12] := 2.209013;
   DATA[502,13] := 978.0345;
   DATA[502,14] := 1.0;
   DATA[502,15] := 2.0;
   DATA[502,16] := 1.0;
   DATA[502,17] := 1.0;
   DATA[502,18] := 1.0;
   DATA[502,19] := 2.0;
   DATA[502,20] := 148.808;
   DATA[502,21] := 155.7293;
   DATA[502,22] := 1.719284;
   DATA[502,23] := 983.2863;
   DATA[502,24] := 2.0;
   DATA[502,25] := 2.0;
   DATA[502,26] := 7.880544;
   DATA[502,27] := 145.091;
   DATA[502,28] := 263.4901;
   DATA[502,29] := 12.22763;
   DATA[502,30] := 1.729172;
   DATA[502,31] := 1.261816;
   DATA[502,32] := 0.7353967;
   DATA[502,33] := 0.3065048;
   DATA[502,34] := 2.0;
   DATA[502,35] := 250.9613;
   DATA[502,36] := 1.730048;
   DATA[502,37] := 189.759;
   DATA[502,38] := 0.000128152;
   DATA[502,39] := 1.0;
   DATA[503,0] := 2.621145;
   DATA[503,1] := 532.5029;
   DATA[503,2] := 2.0;
   DATA[503,3] := 2.0;
   DATA[503,4] := 262.1764;
   DATA[503,5] := 8.393873;
   DATA[503,6] := 327.9159;
   DATA[503,7] := 2.443597;
   DATA[503,8] := 2.0;
   DATA[503,9] := 2.0;
   DATA[503,10] := 2.0;
   DATA[503,11] := 19.70037;
   DATA[503,12] := 2.210037;
   DATA[503,13] := 978.1547;
   DATA[503,14] := 1.0;
   DATA[503,15] := 2.0;
   DATA[503,16] := 1.0;
   DATA[503,17] := 1.0;
   DATA[503,18] := 1.0;
   DATA[503,19] := 2.0;
   DATA[503,20] := 148.808;
   DATA[503,21] := 155.7293;
   DATA[503,22] := 1.71813;
   DATA[503,23] := 983.2479;
   DATA[503,24] := 2.0;
   DATA[503,25] := 2.0;
   DATA[503,26] := 7.880544;
   DATA[503,27] := 145.091;
   DATA[503,28] := 263.4901;
   DATA[503,29] := 12.22763;
   DATA[503,30] := 1.729172;
   DATA[503,31] := 1.272192;
   DATA[503,32] := 0.7353967;
   DATA[503,33] := 0.3065048;
   DATA[503,34] := 2.0;
   DATA[503,35] := 250.9613;
   DATA[503,36] := 1.730048;
   DATA[503,37] := 189.759;
   DATA[503,38] := 0.000128152;
   DATA[503,39] := 1.0;
   DATA[504,0] := 2.646126;
   DATA[504,1] := 532.1889;
   DATA[504,2] := 2.0;
   DATA[504,3] := 2.0;
   DATA[504,4] := 262.1764;
   DATA[504,5] := 8.393873;
   DATA[504,6] := 327.9159;
   DATA[504,7] := 2.443597;
   DATA[504,8] := 2.0;
   DATA[504,9] := 2.0;
   DATA[504,10] := 2.0;
   DATA[504,11] := 19.63634;
   DATA[504,12] := 2.210037;
   DATA[504,13] := 978.5953;
   DATA[504,14] := 1.0;
   DATA[504,15] := 2.0;
   DATA[504,16] := 1.0;
   DATA[504,17] := 1.0;
   DATA[504,18] := 1.0;
   DATA[504,19] := 2.0;
   DATA[504,20] := 148.808;
   DATA[504,21] := 155.7293;
   DATA[504,22] := 1.717361;
   DATA[504,23] := 983.4017;
   DATA[504,24] := 2.0;
   DATA[504,25] := 2.0;
   DATA[504,26] := 7.880544;
   DATA[504,27] := 145.091;
   DATA[504,28] := 263.4901;
   DATA[504,29] := 12.07383;
   DATA[504,30] := 1.729172;
   DATA[504,31] := 1.290765;
   DATA[504,32] := 0.7353967;
   DATA[504,33] := 0.3065048;
   DATA[504,34] := 2.0;
   DATA[504,35] := 250.9613;
   DATA[504,36] := 1.730048;
   DATA[504,37] := 189.759;
   DATA[504,38] := 0.000128152;
   DATA[504,39] := 1.0;
   DATA[505,0] := 2.66214;
   DATA[505,1] := 532.1104;
   DATA[505,2] := 2.0;
   DATA[505,3] := 2.0;
   DATA[505,4] := 262.1764;
   DATA[505,5] := 8.393873;
   DATA[505,6] := 327.9159;
   DATA[505,7] := 2.443597;
   DATA[505,8] := 2.0;
   DATA[505,9] := 2.0;
   DATA[505,10] := 2.0;
   DATA[505,11] := 19.62033;
   DATA[505,12] := 2.212087;
   DATA[505,13] := 978.6754;
   DATA[505,14] := 1.0;
   DATA[505,15] := 2.0;
   DATA[505,16] := 1.0;
   DATA[505,17] := 1.0;
   DATA[505,18] := 1.0;
   DATA[505,19] := 2.0;
   DATA[505,20] := 148.808;
   DATA[505,21] := 155.7293;
   DATA[505,22] := 1.717361;
   DATA[505,23] := 983.517;
   DATA[505,24] := 2.0;
   DATA[505,25] := 2.0;
   DATA[505,26] := 7.880544;
   DATA[505,27] := 145.091;
   DATA[505,28] := 263.4901;
   DATA[505,29] := 12.07383;
   DATA[505,30] := 1.729172;
   DATA[505,31] := 1.291405;
   DATA[505,32] := 0.7353967;
   DATA[505,33] := 0.3065048;
   DATA[505,34] := 2.0;
   DATA[505,35] := 250.9613;
   DATA[505,36] := 1.730048;
   DATA[505,37] := 189.759;
   DATA[505,38] := 0.000128152;
   DATA[505,39] := 1.0;
   DATA[506,0] := 2.66214;
   DATA[506,1] := 532.1889;
   DATA[506,2] := 2.0;
   DATA[506,3] := 2.0;
   DATA[506,4] := 262.1764;
   DATA[506,5] := 8.395155;
   DATA[506,6] := 327.9159;
   DATA[506,7] := 2.443597;
   DATA[506,8] := 2.0;
   DATA[506,9] := 2.0;
   DATA[506,10] := 2.0;
   DATA[506,11] := 19.62033;
   DATA[506,12] := 2.212087;
   DATA[506,13] := 978.9557;
   DATA[506,14] := 1.0;
   DATA[506,15] := 2.0;
   DATA[506,16] := 1.0;
   DATA[506,17] := 1.0;
   DATA[506,18] := 1.0;
   DATA[506,19] := 2.0;
   DATA[506,20] := 148.808;
   DATA[506,21] := 155.7293;
   DATA[506,22] := 1.717361;
   DATA[506,23] := 983.7862;
   DATA[506,24] := 2.0;
   DATA[506,25] := 2.0;
   DATA[506,26] := 7.880544;
   DATA[506,27] := 145.091;
   DATA[506,28] := 263.4901;
   DATA[506,29] := 12.07383;
   DATA[506,30] := 1.725455;
   DATA[506,31] := 1.296529;
   DATA[506,32] := 0.7353967;
   DATA[506,33] := 0.3065048;
   DATA[506,34] := 2.0;
   DATA[506,35] := 250.9613;
   DATA[506,36] := 1.730048;
   DATA[506,37] := 189.6629;
   DATA[506,38] := 0.000128152;
   DATA[506,39] := 1.0;
   DATA[507,0] := 2.634596;
   DATA[507,1] := 531.9926;
   DATA[507,2] := 2.0;
   DATA[507,3] := 2.0;
   DATA[507,4] := 262.1764;
   DATA[507,5] := 8.395475;
   DATA[507,6] := 327.9159;
   DATA[507,7] := 2.443597;
   DATA[507,8] := 2.0;
   DATA[507,9] := 2.0;
   DATA[507,10] := 2.0;
   DATA[507,11] := 19.62033;
   DATA[507,12] := 2.212087;
   DATA[507,13] := 978.7555;
   DATA[507,14] := 1.0;
   DATA[507,15] := 2.0;
   DATA[507,16] := 1.0;
   DATA[507,17] := 1.0;
   DATA[507,18] := 1.0;
   DATA[507,19] := 2.0;
   DATA[507,20] := 148.808;
   DATA[507,21] := 155.8318;
   DATA[507,22] := 1.717361;
   DATA[507,23] := 984.0169;
   DATA[507,24] := 2.0;
   DATA[507,25] := 2.0;
   DATA[507,26] := 7.880544;
   DATA[507,27] := 145.091;
   DATA[507,28] := 263.4901;
   DATA[507,29] := 12.07383;
   DATA[507,30] := 1.724942;
   DATA[507,31] := 1.301652;
   DATA[507,32] := 0.7353967;
   DATA[507,33] := 0.3081703;
   DATA[507,34] := 2.0;
   DATA[507,35] := 250.8171;
   DATA[507,36] := 1.730048;
   DATA[507,37] := 189.5027;
   DATA[507,38] := 0.000128152;
   DATA[507,39] := 1.0;
   DATA[508,0] := 2.621145;
   DATA[508,1] := 532.1104;
   DATA[508,2] := 2.0;
   DATA[508,3] := 2.0;
   DATA[508,4] := 262.1764;
   DATA[508,5] := 8.395475;
   DATA[508,6] := 327.9159;
   DATA[508,7] := 2.441803;
   DATA[508,8] := 2.0;
   DATA[508,9] := 2.0;
   DATA[508,10] := 2.0;
   DATA[508,11] := 19.64594;
   DATA[508,12] := 2.212343;
   DATA[508,13] := 978.7555;
   DATA[508,14] := 1.0;
   DATA[508,15] := 2.0;
   DATA[508,16] := 1.0;
   DATA[508,17] := 1.0;
   DATA[508,18] := 1.0;
   DATA[508,19] := 2.0;
   DATA[508,20] := 148.808;
   DATA[508,21] := 155.96;
   DATA[508,22] := 1.717105;
   DATA[508,23] := 984.2476;
   DATA[508,24] := 2.0;
   DATA[508,25] := 2.0;
   DATA[508,26] := 7.880544;
   DATA[508,27] := 145.091;
   DATA[508,28] := 263.4901;
   DATA[508,29] := 12.07383;
   DATA[508,30] := 1.724942;
   DATA[508,31] := 1.287434;
   DATA[508,32] := 0.7353967;
   DATA[508,33] := 0.3084905;
   DATA[508,34] := 2.0;
   DATA[508,35] := 250.737;
   DATA[508,36] := 1.730048;
   DATA[508,37] := 189.5027;
   DATA[508,38] := 0.000128152;
   DATA[508,39] := 1.0;
   DATA[509,0] := 2.6157;
   DATA[509,1] := 532.1497;
   DATA[509,2] := 2.0;
   DATA[509,3] := 2.0;
   DATA[509,4] := 262.1764;
   DATA[509,5] := 8.395475;
   DATA[509,6] := 327.9159;
   DATA[509,7] := 2.441803;
   DATA[509,8] := 2.0;
   DATA[509,9] := 2.0;
   DATA[509,10] := 2.0;
   DATA[509,11] := 19.66835;
   DATA[509,12] := 2.212343;
   DATA[509,13] := 978.7955;
   DATA[509,14] := 1.0;
   DATA[509,15] := 2.0;
   DATA[509,16] := 1.0;
   DATA[509,17] := 1.0;
   DATA[509,18] := 1.0;
   DATA[509,19] := 2.0;
   DATA[509,20] := 148.808;
   DATA[509,21] := 155.96;
   DATA[509,22] := 1.715952;
   DATA[509,23] := 984.4014;
   DATA[509,24] := 2.0;
   DATA[509,25] := 2.0;
   DATA[509,26] := 7.880544;
   DATA[509,27] := 145.091;
   DATA[509,28] := 263.4901;
   DATA[509,29] := 12.07383;
   DATA[509,30] := 1.724942;
   DATA[509,31] := 1.274753;
   DATA[509,32] := 0.7353967;
   DATA[509,33] := 0.3084905;
   DATA[509,34] := 2.0;
   DATA[509,35] := 250.5928;
   DATA[509,36] := 1.730048;
   DATA[509,37] := 189.4226;
   DATA[509,38] := 0.000128152;
   DATA[509,39] := 1.0;
   DATA[510,0] := 2.6157;
   DATA[510,1] := 531.7178;
   DATA[510,2] := 2.0;
   DATA[510,3] := 2.0;
   DATA[510,4] := 262.1764;
   DATA[510,5] := 8.395475;
   DATA[510,6] := 327.9159;
   DATA[510,7] := 2.441803;
   DATA[510,8] := 2.0;
   DATA[510,9] := 2.0;
   DATA[510,10] := 2.0;
   DATA[510,11] := 19.66835;
   DATA[510,12] := 2.208884;
   DATA[510,13] := 979.3963;
   DATA[510,14] := 1.0;
   DATA[510,15] := 2.0;
   DATA[510,16] := 1.0;
   DATA[510,17] := 1.0;
   DATA[510,18] := 1.0;
   DATA[510,19] := 2.0;
   DATA[510,20] := 148.808;
   DATA[510,21] := 155.96;
   DATA[510,22] := 1.715952;
   DATA[510,23] := 984.4014;
   DATA[510,24] := 2.0;
   DATA[510,25] := 2.0;
   DATA[510,26] := 7.880544;
   DATA[510,27] := 145.091;
   DATA[510,28] := 263.4901;
   DATA[510,29] := 12.07383;
   DATA[510,30] := 1.724942;
   DATA[510,31] := 1.257205;
   DATA[510,32] := 0.7353967;
   DATA[510,33] := 0.3084905;
   DATA[510,34] := 2.0;
   DATA[510,35] := 250.5928;
   DATA[510,36] := 1.730048;
   DATA[510,37] := 189.4226;
   DATA[510,38] := 0.000128152;
   DATA[510,39] := 1.0;
   DATA[511,0] := 2.598085;
   DATA[511,1] := 531.8749;
   DATA[511,2] := 2.0;
   DATA[511,3] := 2.0;
   DATA[511,4] := 262.1764;
   DATA[511,5] := 8.395475;
   DATA[511,6] := 327.9159;
   DATA[511,7] := 2.441803;
   DATA[511,8] := 2.0;
   DATA[511,9] := 2.0;
   DATA[511,10] := 2.0;
   DATA[511,11] := 19.66835;
   DATA[511,12] := 2.208884;
   DATA[511,13] := 980.0372;
   DATA[511,14] := 1.0;
   DATA[511,15] := 2.0;
   DATA[511,16] := 1.0;
   DATA[511,17] := 1.0;
   DATA[511,18] := 1.0;
   DATA[511,19] := 2.0;
   DATA[511,20] := 148.808;
   DATA[511,21] := 155.96;
   DATA[511,22] := 1.715952;
   DATA[511,23] := 984.4783;
   DATA[511,24] := 2.0;
   DATA[511,25] := 2.0;
   DATA[511,26] := 7.880544;
   DATA[511,27] := 144.9628;
   DATA[511,28] := 263.4901;
   DATA[511,29] := 12.07383;
   DATA[511,30] := 1.724942;
   DATA[511,31] := 1.254643;
   DATA[511,32] := 0.7353967;
   DATA[511,33] := 0.3084905;
   DATA[511,34] := 2.0;
   DATA[511,35] := 250.5928;
   DATA[511,36] := 1.730048;
   DATA[511,37] := 189.4226;
   DATA[511,38] := 0.000128152;
   DATA[511,39] := 1.0;
   DATA[512,0] := 2.584953;
   DATA[512,1] := 531.9534;
   DATA[512,2] := 2.0;
   DATA[512,3] := 2.0;
   DATA[512,4] := 262.1764;
   DATA[512,5] := 8.395475;
   DATA[512,6] := 327.9159;
   DATA[512,7] := 2.443597;
   DATA[512,8] := 2.0;
   DATA[512,9] := 2.0;
   DATA[512,10] := 2.0;
   DATA[512,11] := 19.66835;
   DATA[512,12] := 2.208244;
   DATA[512,13] := 980.2775;
   DATA[512,14] := 1.0;
   DATA[512,15] := 2.0;
   DATA[512,16] := 1.0;
   DATA[512,17] := 1.0;
   DATA[512,18] := 1.0;
   DATA[512,19] := 2.0;
   DATA[512,20] := 148.808;
   DATA[512,21] := 155.96;
   DATA[512,22] := 1.715952;
   DATA[512,23] := 984.7475;
   DATA[512,24] := 2.0;
   DATA[512,25] := 2.0;
   DATA[512,26] := 7.880544;
   DATA[512,27] := 144.9628;
   DATA[512,28] := 263.4901;
   DATA[512,29] := 12.07383;
   DATA[512,30] := 1.724942;
   DATA[512,31] := 1.261048;
   DATA[512,32] := 0.7353967;
   DATA[512,33] := 0.3084905;
   DATA[512,34] := 2.0;
   DATA[512,35] := 250.8171;
   DATA[512,36] := 1.730048;
   DATA[512,37] := 189.4226;
   DATA[512,38] := 0.000128152;
   DATA[512,39] := 1.0;
   DATA[513,0] := 2.566057;
   DATA[513,1] := 532.1497;
   DATA[513,2] := 2.0;
   DATA[513,3] := 2.0;
   DATA[513,4] := 262.1764;
   DATA[513,5] := 8.395475;
   DATA[513,6] := 327.9159;
   DATA[513,7] := 2.443982;
   DATA[513,8] := 2.0;
   DATA[513,9] := 2.0;
   DATA[513,10] := 2.0;
   DATA[513,11] := 19.69396;
   DATA[513,12] := 2.207347;
   DATA[513,13] := 979.9971;
   DATA[513,14] := 1.0;
   DATA[513,15] := 2.0;
   DATA[513,16] := 1.0;
   DATA[513,17] := 1.0;
   DATA[513,18] := 1.0;
   DATA[513,19] := 2.0;
   DATA[513,20] := 148.808;
   DATA[513,21] := 155.96;
   DATA[513,22] := 1.715952;
   DATA[513,23] := 984.7475;
   DATA[513,24] := 2.0;
   DATA[513,25] := 2.0;
   DATA[513,26] := 7.880544;
   DATA[513,27] := 144.9628;
   DATA[513,28] := 263.4901;
   DATA[513,29] := 12.07383;
   DATA[513,30] := 1.726352;
   DATA[513,31] := 1.267709;
   DATA[513,32] := 0.7353967;
   DATA[513,33] := 0.3084905;
   DATA[513,34] := 2.0;
   DATA[513,35] := 250.8171;
   DATA[513,36] := 1.730048;
   DATA[513,37] := 189.5668;
   DATA[513,38] := 0.000128152;
   DATA[513,39] := 1.0;
   DATA[514,0] := 2.551645;
   DATA[514,1] := 532.3066;
   DATA[514,2] := 2.0;
   DATA[514,3] := 2.0;
   DATA[514,4] := 262.1764;
   DATA[514,5] := 8.395475;
   DATA[514,6] := 327.9159;
   DATA[514,7] := 2.445007;
   DATA[514,8] := 2.0;
   DATA[514,9] := 2.0;
   DATA[514,10] := 2.0;
   DATA[514,11] := 19.70037;
   DATA[514,12] := 2.207347;
   DATA[514,13] := 980.2375;
   DATA[514,14] := 1.0;
   DATA[514,15] := 2.0;
   DATA[514,16] := 1.0;
   DATA[514,17] := 1.0;
   DATA[514,18] := 1.0;
   DATA[514,19] := 2.0;
   DATA[514,20] := 148.808;
   DATA[514,21] := 155.96;
   DATA[514,22] := 1.717233;
   DATA[514,23] := 984.7475;
   DATA[514,24] := 2.0;
   DATA[514,25] := 2.0;
   DATA[514,26] := 7.880544;
   DATA[514,27] := 144.9628;
   DATA[514,28] := 263.4901;
   DATA[514,29] := 12.07383;
   DATA[514,30] := 1.727634;
   DATA[514,31] := 1.272064;
   DATA[514,32] := 0.7353967;
   DATA[514,33] := 0.3068891;
   DATA[514,34] := 2.0;
   DATA[514,35] := 250.9453;
   DATA[514,36] := 1.730048;
   DATA[514,37] := 189.6469;
   DATA[514,38] := 0.000128152;
   DATA[514,39] := 1.0;
   DATA[515,0] := 2.532108;
   DATA[515,1] := 532.4637;
   DATA[515,2] := 2.0;
   DATA[515,3] := 2.0;
   DATA[515,4] := 262.1764;
   DATA[515,5] := 8.395475;
   DATA[515,6] := 327.9159;
   DATA[515,7] := 2.443085;
   DATA[515,8] := 2.0;
   DATA[515,9] := 2.0;
   DATA[515,10] := 2.0;
   DATA[515,11] := 19.70997;
   DATA[515,12] := 2.206963;
   DATA[515,13] := 980.8383;
   DATA[515,14] := 1.0;
   DATA[515,15] := 2.0;
   DATA[515,16] := 1.0;
   DATA[515,17] := 1.0;
   DATA[515,18] := 1.0;
   DATA[515,19] := 2.0;
   DATA[515,20] := 148.808;
   DATA[515,21] := 155.96;
   DATA[515,22] := 1.717233;
   DATA[515,23] := 984.6706;
   DATA[515,24] := 2.0;
   DATA[515,25] := 2.0;
   DATA[515,26] := 7.880544;
   DATA[515,27] := 144.9628;
   DATA[515,28] := 263.4901;
   DATA[515,29] := 12.07383;
   DATA[515,30] := 1.728275;
   DATA[515,31] := 1.272064;
   DATA[515,32] := 0.7353967;
   DATA[515,33] := 0.3068891;
   DATA[515,34] := 2.0;
   DATA[515,35] := 250.9453;
   DATA[515,36] := 1.730048;
   DATA[515,37] := 189.6949;
   DATA[515,38] := 0.000128152;
   DATA[515,39] := 1.0;
   DATA[516,0] := 2.513211;
   DATA[516,1] := 532.5422;
   DATA[516,2] := 2.0;
   DATA[516,3] := 2.0;
   DATA[516,4] := 262.1764;
   DATA[516,5] := 8.395475;
   DATA[516,6] := 327.9159;
   DATA[516,7] := 2.442828;
   DATA[516,8] := 2.0;
   DATA[516,9] := 2.0;
   DATA[516,10] := 2.0;
   DATA[516,11] := 19.73238;
   DATA[516,12] := 2.209269;
   DATA[516,13] := 980.9985;
   DATA[516,14] := 1.0;
   DATA[516,15] := 2.0;
   DATA[516,16] := 1.0;
   DATA[516,17] := 1.0;
   DATA[516,18] := 1.0;
   DATA[516,19] := 2.0;
   DATA[516,20] := 148.808;
   DATA[516,21] := 155.96;
   DATA[516,22] := 1.717233;
   DATA[516,23] := 984.6706;
   DATA[516,24] := 2.0;
   DATA[516,25] := 2.0;
   DATA[516,26] := 7.880544;
   DATA[516,27] := 144.9628;
   DATA[516,28] := 263.4901;
   DATA[516,29] := 12.07383;
   DATA[516,30] := 1.728275;
   DATA[516,31] := 1.261176;
   DATA[516,32] := 0.7353967;
   DATA[516,33] := 0.3068891;
   DATA[516,34] := 2.0;
   DATA[516,35] := 250.9453;
   DATA[516,36] := 1.585878;
   DATA[516,37] := 189.6949;
   DATA[516,38] := 0.000128152;
   DATA[516,39] := 1.0;
   DATA[517,0] := 2.499439;
   DATA[517,1] := 532.6992;
   DATA[517,2] := 2.0;
   DATA[517,3] := 2.0;
   DATA[517,4] := 262.1764;
   DATA[517,5] := 8.395475;
   DATA[517,6] := 327.9159;
   DATA[517,7] := 2.442828;
   DATA[517,8] := 2.0;
   DATA[517,9] := 2.0;
   DATA[517,10] := 2.0;
   DATA[517,11] := 19.73238;
   DATA[517,12] := 2.209525;
   DATA[517,13] := 981.4391;
   DATA[517,14] := 1.0;
   DATA[517,15] := 2.0;
   DATA[517,16] := 1.0;
   DATA[517,17] := 1.0;
   DATA[517,18] := 1.0;
   DATA[517,19] := 2.0;
   DATA[517,20] := 148.808;
   DATA[517,21] := 155.96;
   DATA[517,22] := 1.717233;
   DATA[517,23] := 985.0167;
   DATA[517,24] := 2.0;
   DATA[517,25] := 2.0;
   DATA[517,26] := 7.880544;
   DATA[517,27] := 144.9628;
   DATA[517,28] := 263.2018;
   DATA[517,29] := 12.07383;
   DATA[517,30] := 1.729172;
   DATA[517,31] := 1.258102;
   DATA[517,32] := 0.7353967;
   DATA[517,33] := 0.3068891;
   DATA[517,34] := 2.0;
   DATA[517,35] := 250.9453;
   DATA[517,36] := 1.585878;
   DATA[517,37] := 189.6949;
   DATA[517,38] := 0.000128152;
   DATA[517,39] := 1.0;
   DATA[518,0] := 2.486628;
   DATA[518,1] := 532.3851;
   DATA[518,2] := 2.0;
   DATA[518,3] := 2.0;
   DATA[518,4] := 262.1764;
   DATA[518,5] := 8.395475;
   DATA[518,6] := 327.9159;
   DATA[518,7] := 2.442828;
   DATA[518,8] := 2.0;
   DATA[518,9] := 2.0;
   DATA[518,10] := 2.0;
   DATA[518,11] := 19.68756;
   DATA[518,12] := 2.209525;
   DATA[518,13] := 981.4391;
   DATA[518,14] := 1.0;
   DATA[518,15] := 2.0;
   DATA[518,16] := 1.0;
   DATA[518,17] := 1.0;
   DATA[518,18] := 1.0;
   DATA[518,19] := 2.0;
   DATA[518,20] := 148.808;
   DATA[518,21] := 155.96;
   DATA[518,22] := 1.717233;
   DATA[518,23] := 985.1705;
   DATA[518,24] := 2.0;
   DATA[518,25] := 2.0;
   DATA[518,26] := 7.880544;
   DATA[518,27] := 144.9628;
   DATA[518,28] := 263.2018;
   DATA[518,29] := 12.07383;
   DATA[518,30] := 1.729172;
   DATA[518,31] := 1.254259;
   DATA[518,32] := 0.7353967;
   DATA[518,33] := 0.3068891;
   DATA[518,34] := 2.0;
   DATA[518,35] := 250.9453;
   DATA[518,36] := 1.730048;
   DATA[518,37] := 189.743;
   DATA[518,38] := 0.000128152;
   DATA[518,39] := 1.0;
   DATA[519,0] := 2.471575;
   DATA[519,1] := 532.4637;
   DATA[519,2] := 2.0;
   DATA[519,3] := 2.0;
   DATA[519,4] := 262.1764;
   DATA[519,5] := 8.395475;
   DATA[519,6] := 327.9159;
   DATA[519,7] := 2.442316;
   DATA[519,8] := 2.0;
   DATA[519,9] := 2.0;
   DATA[519,10] := 2.0;
   DATA[519,11] := 19.67476;
   DATA[519,12] := 2.209525;
   DATA[519,13] := 981.399;
   DATA[519,14] := 1.0;
   DATA[519,15] := 2.0;
   DATA[519,16] := 1.0;
   DATA[519,17] := 1.0;
   DATA[519,18] := 1.0;
   DATA[519,19] := 2.0;
   DATA[519,20] := 148.808;
   DATA[519,21] := 155.96;
   DATA[519,22] := 1.718643;
   DATA[519,23] := 985.0551;
   DATA[519,24] := 2.0;
   DATA[519,25] := 2.0;
   DATA[519,26] := 7.880544;
   DATA[519,27] := 144.9628;
   DATA[519,28] := 263.2018;
   DATA[519,29] := 12.07383;
   DATA[519,30] := 1.729172;
   DATA[519,31] := 1.253875;
   DATA[519,32] := 0.7353967;
   DATA[519,33] := 0.3068891;
   DATA[519,34] := 2.0;
   DATA[519,35] := 250.9453;
   DATA[519,36] := 1.778105;
   DATA[519,37] := 189.743;
   DATA[519,38] := 0.000128152;
   DATA[519,39] := 1.0;
   DATA[520,0] := 2.452679;
   DATA[520,1] := 532.1104;
   DATA[520,2] := 2.0;
   DATA[520,3] := 2.0;
   DATA[520,4] := 262.1764;
   DATA[520,5] := 8.395475;
   DATA[520,6] := 327.9159;
   DATA[520,7] := 2.442188;
   DATA[520,8] := 2.0;
   DATA[520,9] := 2.0;
   DATA[520,10] := 2.0;
   DATA[520,11] := 19.61073;
   DATA[520,12] := 2.209525;
   DATA[520,13] := 981.4391;
   DATA[520,14] := 1.0;
   DATA[520,15] := 2.0;
   DATA[520,16] := 1.0;
   DATA[520,17] := 1.0;
   DATA[520,18] := 1.0;
   DATA[520,19] := 2.0;
   DATA[520,20] := 148.808;
   DATA[520,21] := 155.96;
   DATA[520,22] := 1.720053;
   DATA[520,23] := 984.8244;
   DATA[520,24] := 2.0;
   DATA[520,25] := 2.0;
   DATA[520,26] := 7.880544;
   DATA[520,27] := 144.9628;
   DATA[520,28] := 263.2018;
   DATA[520,29] := 12.07383;
   DATA[520,30] := 1.729172;
   DATA[520,31] := 1.268733;
   DATA[520,32] := 0.7353967;
   DATA[520,33] := 0.3068891;
   DATA[520,34] := 2.0;
   DATA[520,35] := 250.9453;
   DATA[520,36] := 1.681991;
   DATA[520,37] := 189.743;
   DATA[520,38] := 0.000128152;
   DATA[520,39] := 1.0;
   DATA[521,0] := 2.438267;
   DATA[521,1] := 532.2674;
   DATA[521,2] := 2.0;
   DATA[521,3] := 2.0;
   DATA[521,4] := 262.1764;
   DATA[521,5] := 8.395475;
   DATA[521,6] := 327.9159;
   DATA[521,7] := 2.442188;
   DATA[521,8] := 2.0;
   DATA[521,9] := 2.0;
   DATA[521,10] := 2.0;
   DATA[521,11] := 19.55631;
   DATA[521,12] := 2.209525;
   DATA[521,13] := 981.9598;
   DATA[521,14] := 1.0;
   DATA[521,15] := 2.0;
   DATA[521,16] := 1.0;
   DATA[521,17] := 1.0;
   DATA[521,18] := 1.0;
   DATA[521,19] := 2.0;
   DATA[521,20] := 148.808;
   DATA[521,21] := 155.96;
   DATA[521,22] := 1.720565;
   DATA[521,23] := 984.9782;
   DATA[521,24] := 2.0;
   DATA[521,25] := 2.0;
   DATA[521,26] := 7.880544;
   DATA[521,27] := 144.9628;
   DATA[521,28] := 263.4901;
   DATA[521,29] := 12.07383;
   DATA[521,30] := 1.729172;
   DATA[521,31] := 1.279749;
   DATA[521,32] := 0.7353967;
   DATA[521,33] := 0.3064407;
   DATA[521,34] := 2.0;
   DATA[521,35] := 251.1215;
   DATA[521,36] := 1.681991;
   DATA[521,37] := 189.743;
   DATA[521,38] := 0.000128152;
   DATA[521,39] := 1.0;
   DATA[522,0] := 2.425776;
   DATA[522,1] := 532.2674;
   DATA[522,2] := 2.0;
   DATA[522,3] := 2.0;
   DATA[522,4] := 262.1764;
   DATA[522,5] := 8.395475;
   DATA[522,6] := 327.9159;
   DATA[522,7] := 2.442956;
   DATA[522,8] := 2.0;
   DATA[522,9] := 2.0;
   DATA[522,10] := 2.0;
   DATA[522,11] := 19.54671;
   DATA[522,12] := 2.209525;
   DATA[522,13] := 982.3603;
   DATA[522,14] := 1.0;
   DATA[522,15] := 2.0;
   DATA[522,16] := 1.0;
   DATA[522,17] := 1.0;
   DATA[522,18] := 1.0;
   DATA[522,19] := 2.0;
   DATA[522,20] := 148.808;
   DATA[522,21] := 155.8318;
   DATA[522,22] := 1.720565;
   DATA[522,23] := 984.7475;
   DATA[522,24] := 2.0;
   DATA[522,25] := 2.0;
   DATA[522,26] := 7.880544;
   DATA[522,27] := 144.9628;
   DATA[522,28] := 263.4901;
   DATA[522,29] := 12.07383;
   DATA[522,30] := 1.729172;
   DATA[522,31] := 1.281158;
   DATA[522,32] := 0.7353967;
   DATA[522,33] := 0.3064407;
   DATA[522,34] := 2.0;
   DATA[522,35] := 251.2176;
   DATA[522,36] := 1.681991;
   DATA[522,37] := 189.743;
   DATA[522,38] := 0.000128152;
   DATA[522,39] := 1.0;
   DATA[523,0] := 2.422573;
   DATA[523,1] := 532.1497;
   DATA[523,2] := 2.0;
   DATA[523,3] := 2.0;
   DATA[523,4] := 262.1764;
   DATA[523,5] := 8.395475;
   DATA[523,6] := 327.9159;
   DATA[523,7] := 2.444623;
   DATA[523,8] := 2.0;
   DATA[523,9] := 2.0;
   DATA[523,10] := 2.0;
   DATA[523,11] := 19.54671;
   DATA[523,12] := 2.209525;
   DATA[523,13] := 982.16;
   DATA[523,14] := 1.0;
   DATA[523,15] := 2.0;
   DATA[523,16] := 1.0;
   DATA[523,17] := 1.0;
   DATA[523,18] := 1.0;
   DATA[523,19] := 2.0;
   DATA[523,20] := 148.808;
   DATA[523,21] := 155.8318;
   DATA[523,22] := 1.720565;
   DATA[523,23] := 984.7859;
   DATA[523,24] := 2.0;
   DATA[523,25] := 2.0;
   DATA[523,26] := 7.880544;
   DATA[523,27] := 144.9628;
   DATA[523,28] := 263.4901;
   DATA[523,29] := 12.07383;
   DATA[523,30] := 1.730069;
   DATA[523,31] := 1.275906;
   DATA[523,32] := 0.7353967;
   DATA[523,33] := 0.3064407;
   DATA[523,34] := 2.0;
   DATA[523,35] := 251.2337;
   DATA[523,36] := 1.681991;
   DATA[523,37] := 189.743;
   DATA[523,38] := 0.000128152;
   DATA[523,39] := 1.0;
   DATA[524,0] := 2.422573;
   DATA[524,1] := 531.8749;
   DATA[524,2] := 2.0;
   DATA[524,3] := 2.0;
   DATA[524,4] := 262.1764;
   DATA[524,5] := 8.395475;
   DATA[524,6] := 327.9159;
   DATA[524,7] := 2.445519;
   DATA[524,8] := 2.0;
   DATA[524,9] := 2.0;
   DATA[524,10] := 2.0;
   DATA[524,11] := 19.57872;
   DATA[524,12] := 2.209525;
   DATA[524,13] := 982.4004;
   DATA[524,14] := 1.0;
   DATA[524,15] := 2.0;
   DATA[524,16] := 1.0;
   DATA[524,17] := 1.0;
   DATA[524,18] := 1.0;
   DATA[524,19] := 2.0;
   DATA[524,20] := 148.808;
   DATA[524,21] := 155.8318;
   DATA[524,22] := 1.720565;
   DATA[524,23] := 984.6706;
   DATA[524,24] := 2.0;
   DATA[524,25] := 2.0;
   DATA[524,26] := 7.880544;
   DATA[524,27] := 144.9628;
   DATA[524,28] := 263.4901;
   DATA[524,29] := 12.07383;
   DATA[524,30] := 1.730838;
   DATA[524,31] := 1.275906;
   DATA[524,32] := 0.7353967;
   DATA[524,33] := 0.3070813;
   DATA[524,34] := 2.0;
   DATA[524,35] := 251.2337;
   DATA[524,36] := 1.681991;
   DATA[524,37] := 189.9353;
   DATA[524,38] := 0.000128152;
   DATA[524,39] := 1.0;
   DATA[525,0] := 2.463889;
   DATA[525,1] := 531.0898;
   DATA[525,2] := 2.0;
   DATA[525,3] := 2.0;
   DATA[525,4] := 262.1764;
   DATA[525,5] := 8.395475;
   DATA[525,6] := 327.9159;
   DATA[525,7] := 2.445519;
   DATA[525,8] := 2.0;
   DATA[525,9] := 2.0;
   DATA[525,10] := 2.0;
   DATA[525,11] := 19.58192;
   DATA[525,12] := 2.209525;
   DATA[525,13] := 982.4004;
   DATA[525,14] := 1.0;
   DATA[525,15] := 2.0;
   DATA[525,16] := 1.0;
   DATA[525,17] := 1.0;
   DATA[525,18] := 1.0;
   DATA[525,19] := 2.0;
   DATA[525,20] := 148.808;
   DATA[525,21] := 155.8318;
   DATA[525,22] := 1.720565;
   DATA[525,23] := 984.7475;
   DATA[525,24] := 2.0;
   DATA[525,25] := 2.0;
   DATA[525,26] := 7.880544;
   DATA[525,27] := 144.9628;
   DATA[525,28] := 263.4901;
   DATA[525,29] := 12.07383;
   DATA[525,30] := 1.730838;
   DATA[525,31] := 1.26361;
   DATA[525,32] := 0.7353967;
   DATA[525,33] := 0.3070813;
   DATA[525,34] := 2.0;
   DATA[525,35] := 251.2337;
   DATA[525,36] := 1.730048;
   DATA[525,37] := 189.9833;
   DATA[525,38] := 0.000128152;
   DATA[525,39] := 1.0;
   DATA[526,0] := 2.514493;
   DATA[526,1] := 530.7365;
   DATA[526,2] := 2.0;
   DATA[526,3] := 2.0;
   DATA[526,4] := 262.1764;
   DATA[526,5] := 8.395475;
   DATA[526,6] := 327.9159;
   DATA[526,7] := 2.445519;
   DATA[526,8] := 2.0;
   DATA[526,9] := 2.0;
   DATA[526,10] := 2.0;
   DATA[526,11] := 19.58832;
   DATA[526,12] := 2.209525;
   DATA[526,13] := 982.5606;
   DATA[526,14] := 1.0;
   DATA[526,15] := 2.0;
   DATA[526,16] := 1.0;
   DATA[526,17] := 1.0;
   DATA[526,18] := 1.0;
   DATA[526,19] := 2.0;
   DATA[526,20] := 148.808;
   DATA[526,21] := 155.8318;
   DATA[526,22] := 1.720565;
   DATA[526,23] := 984.6321;
   DATA[526,24] := 2.0;
   DATA[526,25] := 2.0;
   DATA[526,26] := 7.880544;
   DATA[526,27] := 144.9628;
   DATA[526,28] := 263.4901;
   DATA[526,29] := 12.07383;
   DATA[526,30] := 1.730838;
   DATA[526,31] := 1.261432;
   DATA[526,32] := 0.7353967;
   DATA[526,33] := 0.3070813;
   DATA[526,34] := 2.0;
   DATA[526,35] := 251.2337;
   DATA[526,36] := 1.730048;
   DATA[526,37] := 189.9833;
   DATA[526,38] := 0.000128152;
   DATA[526,39] := 1.0;
   DATA[527,0] := 2.537552;
   DATA[527,1] := 530.5795;
   DATA[527,2] := 2.0;
   DATA[527,3] := 2.0;
   DATA[527,4] := 262.1764;
   DATA[527,5] := 8.395475;
   DATA[527,6] := 327.9159;
   DATA[527,7] := 2.445519;
   DATA[527,8] := 2.0;
   DATA[527,9] := 2.0;
   DATA[527,10] := 2.0;
   DATA[527,11] := 19.58832;
   DATA[527,12] := 2.209525;
   DATA[527,13] := 982.4004;
   DATA[527,14] := 1.0;
   DATA[527,15] := 2.0;
   DATA[527,16] := 1.0;
   DATA[527,17] := 1.0;
   DATA[527,18] := 1.0;
   DATA[527,19] := 2.0;
   DATA[527,20] := 148.808;
   DATA[527,21] := 155.8318;
   DATA[527,22] := 1.720565;
   DATA[527,23] := 984.5552;
   DATA[527,24] := 2.0;
   DATA[527,25] := 2.0;
   DATA[527,26] := 7.880544;
   DATA[527,27] := 144.9628;
   DATA[527,28] := 263.4901;
   DATA[527,29] := 12.07383;
   DATA[527,30] := 1.730838;
   DATA[527,31] := 1.266428;
   DATA[527,32] := 0.7353967;
   DATA[527,33] := 0.3070813;
   DATA[527,34] := 2.0;
   DATA[527,35] := 251.2337;
   DATA[527,36] := 1.810143;
   DATA[527,37] := 189.9833;
   DATA[527,38] := 0.000128152;
   DATA[527,39] := 1.0;
   DATA[528,0] := 2.583352;
   DATA[528,1] := 530.3832;
   DATA[528,2] := 2.0;
   DATA[528,3] := 2.0;
   DATA[528,4] := 262.1764;
   DATA[528,5] := 8.395475;
   DATA[528,6] := 327.9159;
   DATA[528,7] := 2.445519;
   DATA[528,8] := 2.0;
   DATA[528,9] := 2.0;
   DATA[528,10] := 2.0;
   DATA[528,11] := 19.58832;
   DATA[528,12] := 2.209525;
   DATA[528,13] := 982.4004;
   DATA[528,14] := 1.0;
   DATA[528,15] := 2.0;
   DATA[528,16] := 1.0;
   DATA[528,17] := 1.0;
   DATA[528,18] := 1.0;
   DATA[528,19] := 2.0;
   DATA[528,20] := 148.808;
   DATA[528,21] := 155.9087;
   DATA[528,22] := 1.718515;
   DATA[528,23] := 984.4399;
   DATA[528,24] := 2.0;
   DATA[528,25] := 2.0;
   DATA[528,26] := 7.880544;
   DATA[528,27] := 144.9628;
   DATA[528,28] := 263.4901;
   DATA[528,29] := 12.07383;
   DATA[528,30] := 1.729172;
   DATA[528,31] := 1.266428;
   DATA[528,32] := 0.7353967;
   DATA[528,33] := 0.3070813;
   DATA[528,34] := 2.0;
   DATA[528,35] := 251.2657;
   DATA[528,36] := 1.810143;
   DATA[528,37] := 189.9833;
   DATA[528,38] := 0.000128152;
   DATA[528,39] := 1.0;
   DATA[529,0] := 2.6157;
   DATA[529,1] := 530.3832;
   DATA[529,2] := 2.0;
   DATA[529,3] := 2.0;
   DATA[529,4] := 262.1764;
   DATA[529,5] := 8.395475;
   DATA[529,6] := 327.9159;
   DATA[529,7] := 2.445519;
   DATA[529,8] := 2.0;
   DATA[529,9] := 2.0;
   DATA[529,10] := 2.0;
   DATA[529,11] := 19.62674;
   DATA[529,12] := 2.209525;
   DATA[529,13] := 982.4805;
   DATA[529,14] := 1.0;
   DATA[529,15] := 2.0;
   DATA[529,16] := 1.0;
   DATA[529,17] := 1.0;
   DATA[529,18] := 1.0;
   DATA[529,19] := 2.0;
   DATA[529,20] := 148.808;
   DATA[529,21] := 155.9087;
   DATA[529,22] := 1.718515;
   DATA[529,23] := 984.4783;
   DATA[529,24] := 2.0;
   DATA[529,25] := 2.0;
   DATA[529,26] := 7.880544;
   DATA[529,27] := 144.9628;
   DATA[529,28] := 263.4901;
   DATA[529,29] := 12.07383;
   DATA[529,30] := 1.728275;
   DATA[529,31] := 1.28372;
   DATA[529,32] := 0.7353967;
   DATA[529,33] := 0.3070813;
   DATA[529,34] := 2.0;
   DATA[529,35] := 251.2657;
   DATA[529,36] := 1.810143;
   DATA[529,37] := 189.9833;
   DATA[529,38] := 0.000128152;
   DATA[529,39] := 1.0;
   DATA[530,0] := 2.644525;
   DATA[530,1] := 530.9328;
   DATA[530,2] := 2.0;
   DATA[530,3] := 2.0;
   DATA[530,4] := 262.1764;
   DATA[530,5] := 8.395475;
   DATA[530,6] := 327.8647;
   DATA[530,7] := 2.445519;
   DATA[530,8] := 2.0;
   DATA[530,9] := 2.0;
   DATA[530,10] := 2.0;
   DATA[530,11] := 19.65875;
   DATA[530,12] := 2.209525;
   DATA[530,13] := 982.2802;
   DATA[530,14] := 1.0;
   DATA[530,15] := 2.0;
   DATA[530,16] := 1.0;
   DATA[530,17] := 1.0;
   DATA[530,18] := 1.0;
   DATA[530,19] := 2.0;
   DATA[530,20] := 148.808;
   DATA[530,21] := 155.9087;
   DATA[530,22] := 1.717746;
   DATA[530,23] := 983.9785;
   DATA[530,24] := 2.0;
   DATA[530,25] := 2.0;
   DATA[530,26] := 7.880544;
   DATA[530,27] := 144.9628;
   DATA[530,28] := 263.4901;
   DATA[530,29] := 12.07383;
   DATA[530,30] := 1.728275;
   DATA[530,31] := 1.298834;
   DATA[530,32] := 0.7353967;
   DATA[530,33] := 0.3065689;
   DATA[530,34] := 2.0;
   DATA[530,35] := 251.2657;
   DATA[530,36] := 1.810143;
   DATA[530,37] := 189.9833;
   DATA[530,38] := 0.000128152;
   DATA[530,39] := 1.0;
   DATA[531,0] := 2.657016;
   DATA[531,1] := 531.2861;
   DATA[531,2] := 2.0;
   DATA[531,3] := 2.0;
   DATA[531,4] := 262.1764;
   DATA[531,5] := 8.395475;
   DATA[531,6] := 327.7108;
   DATA[531,7] := 2.444366;
   DATA[531,8] := 2.0;
   DATA[531,9] := 2.0;
   DATA[531,10] := 2.0;
   DATA[531,11] := 19.65875;
   DATA[531,12] := 2.209525;
   DATA[531,13] := 981.9598;
   DATA[531,14] := 1.0;
   DATA[531,15] := 2.0;
   DATA[531,16] := 1.0;
   DATA[531,17] := 1.0;
   DATA[531,18] := 1.0;
   DATA[531,19] := 2.0;
   DATA[531,20] := 148.808;
   DATA[531,21] := 155.9087;
   DATA[531,22] := 1.717746;
   DATA[531,23] := 984.0169;
   DATA[531,24] := 2.0;
   DATA[531,25] := 2.0;
   DATA[531,26] := 7.880544;
   DATA[531,27] := 144.9628;
   DATA[531,28] := 263.3299;
   DATA[531,29] := 12.07383;
   DATA[531,30] := 1.728275;
   DATA[531,31] := 1.309722;
   DATA[531,32] := 0.7353967;
   DATA[531,33] := 0.3065689;
   DATA[531,34] := 2.0;
   DATA[531,35] := 251.2657;
   DATA[531,36] := 1.778105;
   DATA[531,37] := 189.9833;
   DATA[531,38] := 0.000128152;
   DATA[531,39] := 1.0;
   DATA[532,0] := 2.660859;
   DATA[532,1] := 531.3253;
   DATA[532,2] := 2.0;
   DATA[532,3] := 2.0;
   DATA[532,4] := 262.1764;
   DATA[532,5] := 8.395475;
   DATA[532,6] := 327.7108;
   DATA[532,7] := 2.444366;
   DATA[532,8] := 2.0;
   DATA[532,9] := 2.0;
   DATA[532,10] := 2.0;
   DATA[532,11] := 19.65875;
   DATA[532,12] := 2.209525;
   DATA[532,13] := 981.7595;
   DATA[532,14] := 1.0;
   DATA[532,15] := 2.0;
   DATA[532,16] := 1.0;
   DATA[532,17] := 1.0;
   DATA[532,18] := 1.0;
   DATA[532,19] := 2.0;
   DATA[532,20] := 148.808;
   DATA[532,21] := 155.9344;
   DATA[532,22] := 1.717746;
   DATA[532,23] := 983.8246;
   DATA[532,24] := 2.0;
   DATA[532,25] := 2.0;
   DATA[532,26] := 7.880544;
   DATA[532,27] := 145.1679;
   DATA[532,28] := 263.2658;
   DATA[532,29] := 12.07383;
   DATA[532,30] := 1.726224;
   DATA[532,31] := 1.311003;
   DATA[532,32] := 0.7353967;
   DATA[532,33] := 0.3065689;
   DATA[532,34] := 2.0;
   DATA[532,35] := 251.2657;
   DATA[532,36] := 1.601897;
   DATA[532,37] := 189.9833;
   DATA[532,38] := 0.000128152;
   DATA[532,39] := 1.0;
   DATA[533,0] := 2.646767;
   DATA[533,1] := 531.4824;
   DATA[533,2] := 2.0;
   DATA[533,3] := 2.0;
   DATA[533,4] := 262.1764;
   DATA[533,5] := 8.395475;
   DATA[533,6] := 327.7108;
   DATA[533,7] := 2.444366;
   DATA[533,8] := 2.0;
   DATA[533,9] := 2.0;
   DATA[533,10] := 2.0;
   DATA[533,11] := 19.65875;
   DATA[533,12] := 2.209525;
   DATA[533,13] := 981.5993;
   DATA[533,14] := 1.0;
   DATA[533,15] := 2.0;
   DATA[533,16] := 1.0;
   DATA[533,17] := 1.0;
   DATA[533,18] := 1.0;
   DATA[533,19] := 2.0;
   DATA[533,20] := 148.808;
   DATA[533,21] := 155.9344;
   DATA[533,22] := 1.718771;
   DATA[533,23] := 984.0554;
   DATA[533,24] := 2.0;
   DATA[533,25] := 2.0;
   DATA[533,26] := 7.880544;
   DATA[533,27] := 145.1679;
   DATA[533,28] := 263.2658;
   DATA[533,29] := 12.07383;
   DATA[533,30] := 1.726224;
   DATA[533,31] := 1.301396;
   DATA[533,32] := 0.7353967;
   DATA[533,33] := 0.3065689;
   DATA[533,34] := 2.0;
   DATA[533,35] := 251.2657;
   DATA[533,36] := 1.601897;
   DATA[533,37] := 189.9833;
   DATA[533,38] := 0.000128152;
   DATA[533,39] := 1.0;
   DATA[534,0] := 2.62755;
   DATA[534,1] := 531.4038;
   DATA[534,2] := 2.0;
   DATA[534,3] := 2.0;
   DATA[534,4] := 262.1764;
   DATA[534,5] := 8.395475;
   DATA[534,6] := 327.7108;
   DATA[534,7] := 2.444366;
   DATA[534,8] := 2.0;
   DATA[534,9] := 2.0;
   DATA[534,10] := 2.0;
   DATA[534,11] := 19.70037;
   DATA[534,12] := 2.209525;
   DATA[534,13] := 981.3589;
   DATA[534,14] := 1.0;
   DATA[534,15] := 2.0;
   DATA[534,16] := 1.0;
   DATA[534,17] := 1.0;
   DATA[534,18] := 1.0;
   DATA[534,19] := 2.0;
   DATA[534,20] := 148.808;
   DATA[534,21] := 155.9344;
   DATA[534,22] := 1.721847;
   DATA[534,23] := 983.517;
   DATA[534,24] := 2.0;
   DATA[534,25] := 2.0;
   DATA[534,26] := 7.880544;
   DATA[534,27] := 145.1679;
   DATA[534,28] := 263.2658;
   DATA[534,29] := 12.07383;
   DATA[534,30] := 1.726224;
   DATA[534,31] := 1.29307;
   DATA[534,32] := 0.7353967;
   DATA[534,33] := 0.3065689;
   DATA[534,34] := 2.0;
   DATA[534,35] := 251.2657;
   DATA[534,36] := 1.746067;
   DATA[534,37] := 189.9833;
   DATA[534,38] := 0.000128152;
   DATA[534,39] := 1.0;
   DATA[535,0] := 2.619543;
   DATA[535,1] := 531.4824;
   DATA[535,2] := 2.0;
   DATA[535,3] := 2.0;
   DATA[535,4] := 262.1764;
   DATA[535,5] := 8.395475;
   DATA[535,6] := 327.7108;
   DATA[535,7] := 2.440906;
   DATA[535,8] := 2.0;
   DATA[535,9] := 2.0;
   DATA[535,10] := 2.0;
   DATA[535,11] := 19.72598;
   DATA[535,12] := 2.209525;
   DATA[535,13] := 981.0385;
   DATA[535,14] := 1.0;
   DATA[535,15] := 2.0;
   DATA[535,16] := 1.0;
   DATA[535,17] := 1.0;
   DATA[535,18] := 1.0;
   DATA[535,19] := 2.0;
   DATA[535,20] := 148.808;
   DATA[535,21] := 155.9344;
   DATA[535,22] := 1.722231;
   DATA[535,23] := 983.4786;
   DATA[535,24] := 2.0;
   DATA[535,25] := 2.0;
   DATA[535,26] := 7.880544;
   DATA[535,27] := 144.9628;
   DATA[535,28] := 263.2658;
   DATA[535,29] := 12.07383;
   DATA[535,30] := 1.728531;
   DATA[535,31] := 1.291533;
   DATA[535,32] := 0.7353967;
   DATA[535,33] := 0.3065689;
   DATA[535,34] := 2.0;
   DATA[535,35] := 251.2657;
   DATA[535,36] := 1.746067;
   DATA[535,37] := 189.9353;
   DATA[535,38] := 0.000128152;
   DATA[535,39] := 1.0;
   DATA[536,0] := 2.613778;
   DATA[536,1] := 531.9534;
   DATA[536,2] := 2.0;
   DATA[536,3] := 2.0;
   DATA[536,4] := 262.1764;
   DATA[536,5] := 8.395475;
   DATA[536,6] := 327.7108;
   DATA[536,7] := 2.440137;
   DATA[536,8] := 2.0;
   DATA[536,9] := 2.0;
   DATA[536,10] := 2.0;
   DATA[536,11] := 19.72598;
   DATA[536,12] := 2.209525;
   DATA[536,13] := 980.8783;
   DATA[536,14] := 1.0;
   DATA[536,15] := 2.0;
   DATA[536,16] := 1.0;
   DATA[536,17] := 1.0;
   DATA[536,18] := 1.0;
   DATA[536,19] := 2.0;
   DATA[536,20] := 148.808;
   DATA[536,21] := 155.9344;
   DATA[536,22] := 1.722231;
   DATA[536,23] := 983.4401;
   DATA[536,24] := 2.0;
   DATA[536,25] := 2.0;
   DATA[536,26] := 7.880544;
   DATA[536,27] := 144.9628;
   DATA[536,28] := 263.2658;
   DATA[536,29] := 12.07383;
   DATA[536,30] := 1.728531;
   DATA[536,31] := 1.27834;
   DATA[536,32] := 0.7353967;
   DATA[536,33] := 0.3065689;
   DATA[536,34] := 2.0;
   DATA[536,35] := 251.1375;
   DATA[536,36] := 1.746067;
   DATA[536,37] := 189.8872;
   DATA[536,38] := 0.000128152;
   DATA[536,39] := 1.0;
   DATA[537,0] := 2.602569;
   DATA[537,1] := 531.9141;
   DATA[537,2] := 2.0;
   DATA[537,3] := 2.0;
   DATA[537,4] := 262.1764;
   DATA[537,5] := 8.395475;
   DATA[537,6] := 327.7108;
   DATA[537,7] := 2.439753;
   DATA[537,8] := 2.0;
   DATA[537,9] := 2.0;
   DATA[537,10] := 2.0;
   DATA[537,11] := 19.76759;
   DATA[537,12] := 2.209525;
   DATA[537,13] := 980.8783;
   DATA[537,14] := 1.0;
   DATA[537,15] := 2.0;
   DATA[537,16] := 1.0;
   DATA[537,17] := 1.0;
   DATA[537,18] := 1.0;
   DATA[537,19] := 2.0;
   DATA[537,20] := 148.808;
   DATA[537,21] := 155.9344;
   DATA[537,22] := 1.722231;
   DATA[537,23] := 983.517;
   DATA[537,24] := 2.0;
   DATA[537,25] := 2.0;
   DATA[537,26] := 7.880544;
   DATA[537,27] := 144.9628;
   DATA[537,28] := 263.4581;
   DATA[537,29] := 12.07383;
   DATA[537,30] := 1.7293;
   DATA[537,31] := 1.271679;
   DATA[537,32] := 0.7353967;
   DATA[537,33] := 0.3065689;
   DATA[537,34] := 2.0;
   DATA[537,35] := 251.0254;
   DATA[537,36] := 1.746067;
   DATA[537,37] := 189.8872;
   DATA[537,38] := 0.000128152;
   DATA[537,39] := 1.0;
   DATA[538,0] := 2.580149;
   DATA[538,1] := 532.3066;
   DATA[538,2] := 2.0;
   DATA[538,3] := 2.0;
   DATA[538,4] := 262.1764;
   DATA[538,5] := 8.395475;
   DATA[538,6] := 327.839;
   DATA[538,7] := 2.439753;
   DATA[538,8] := 2.0;
   DATA[538,9] := 2.0;
   DATA[538,10] := 2.0;
   DATA[538,11] := 19.77079;
   DATA[538,12] := 2.21119;
   DATA[538,13] := 980.7582;
   DATA[538,14] := 1.0;
   DATA[538,15] := 2.0;
   DATA[538,16] := 1.0;
   DATA[538,17] := 1.0;
   DATA[538,18] := 1.0;
   DATA[538,19] := 2.0;
   DATA[538,20] := 148.808;
   DATA[538,21] := 155.9344;
   DATA[538,22] := 1.722231;
   DATA[538,23] := 983.4017;
   DATA[538,24] := 2.0;
   DATA[538,25] := 2.0;
   DATA[538,26] := 7.880544;
   DATA[538,27] := 144.9628;
   DATA[538,28] := 263.4581;
   DATA[538,29] := 12.07383;
   DATA[538,30] := 1.7293;
   DATA[538,31] := 1.274241;
   DATA[538,32] := 0.7353967;
   DATA[538,33] := 0.3065689;
   DATA[538,34] := 2.0;
   DATA[538,35] := 251.0254;
   DATA[538,36] := 1.746067;
   DATA[538,37] := 189.8872;
   DATA[538,38] := 0.000128152;
   DATA[538,39] := 1.0;
   DATA[539,0] := 2.567338;
   DATA[539,1] := 532.7384;
   DATA[539,2] := 2.0;
   DATA[539,3] := 2.0;
   DATA[539,4] := 262.1764;
   DATA[539,5] := 8.395475;
   DATA[539,6] := 327.839;
   DATA[539,7] := 2.439753;
   DATA[539,8] := 2.0;
   DATA[539,9] := 2.0;
   DATA[539,10] := 2.0;
   DATA[539,11] := 19.77399;
   DATA[539,12] := 2.21119;
   DATA[539,13] := 980.8783;
   DATA[539,14] := 1.0;
   DATA[539,15] := 2.0;
   DATA[539,16] := 1.0;
   DATA[539,17] := 1.0;
   DATA[539,18] := 1.0;
   DATA[539,19] := 2.0;
   DATA[539,20] := 148.808;
   DATA[539,21] := 155.9344;
   DATA[539,22] := 1.72095;
   DATA[539,23] := 983.5939;
   DATA[539,24] := 2.0;
   DATA[539,25] := 2.0;
   DATA[539,26] := 7.880544;
   DATA[539,27] := 144.9628;
   DATA[539,28] := 263.4581;
   DATA[539,29] := 12.07383;
   DATA[539,30] := 1.7293;
   DATA[539,31] := 1.278724;
   DATA[539,32] := 0.7353967;
   DATA[539,33] := 0.3065689;
   DATA[539,34] := 2.0;
   DATA[539,35] := 251.0254;
   DATA[539,36] := 1.746067;
   DATA[539,37] := 189.8872;
   DATA[539,38] := 0.000128152;
   DATA[539,39] := 1.0;
   DATA[540,0] := 2.551324;
   DATA[540,1] := 533.3665;
   DATA[540,2] := 2.0;
   DATA[540,3] := 2.0;
   DATA[540,4] := 262.1764;
   DATA[540,5] := 8.395475;
   DATA[540,6] := 327.839;
   DATA[540,7] := 2.439753;
   DATA[540,8] := 2.0;
   DATA[540,9] := 2.0;
   DATA[540,10] := 2.0;
   DATA[540,11] := 19.77399;
   DATA[540,12] := 2.21119;
   DATA[540,13] := 980.598;
   DATA[540,14] := 1.0;
   DATA[540,15] := 2.0;
   DATA[540,16] := 1.0;
   DATA[540,17] := 1.0;
   DATA[540,18] := 1.0;
   DATA[540,19] := 2.0;
   DATA[540,20] := 148.808;
   DATA[540,21] := 155.9344;
   DATA[540,22] := 1.72095;
   DATA[540,23] := 983.6708;
   DATA[540,24] := 2.0;
   DATA[540,25] := 2.0;
   DATA[540,26] := 7.880544;
   DATA[540,27] := 144.9628;
   DATA[540,28] := 263.4581;
   DATA[540,29] := 12.07383;
   DATA[540,30] := 1.73071;
   DATA[540,31] := 1.275778;
   DATA[540,32] := 0.7353967;
   DATA[540,33] := 0.3065689;
   DATA[540,34] := 2.0;
   DATA[540,35] := 251.0254;
   DATA[540,36] := 1.746067;
   DATA[540,37] := 189.8872;
   DATA[540,38] := 0.000128152;
   DATA[540,39] := 1.0;
   DATA[541,0] := 2.535951;
   DATA[541,1] := 533.7197;
   DATA[541,2] := 2.0;
   DATA[541,3] := 2.0;
   DATA[541,4] := 262.1764;
   DATA[541,5] := 8.395475;
   DATA[541,6] := 327.839;
   DATA[541,7] := 2.439753;
   DATA[541,8] := 2.0;
   DATA[541,9] := 2.0;
   DATA[541,10] := 2.0;
   DATA[541,11] := 19.77399;
   DATA[541,12] := 2.214009;
   DATA[541,13] := 980.7582;
   DATA[541,14] := 1.0;
   DATA[541,15] := 2.0;
   DATA[541,16] := 1.0;
   DATA[541,17] := 1.0;
   DATA[541,18] := 1.0;
   DATA[541,19] := 2.0;
   DATA[541,20] := 148.808;
   DATA[541,21] := 155.9344;
   DATA[541,22] := 1.72095;
   DATA[541,23] := 983.7093;
   DATA[541,24] := 2.0;
   DATA[541,25] := 2.0;
   DATA[541,26] := 7.87766;
   DATA[541,27] := 144.9628;
   DATA[541,28] := 263.4581;
   DATA[541,29] := 12.07383;
   DATA[541,30] := 1.730838;
   DATA[541,31] := 1.290893;
   DATA[541,32] := 0.7353967;
   DATA[541,33] := 0.3065689;
   DATA[541,34] := 2.0;
   DATA[541,35] := 251.0254;
   DATA[541,36] := 1.746067;
   DATA[541,37] := 189.8872;
   DATA[541,38] := 0.000128152;
   DATA[541,39] := 1.0;
   DATA[542,0] := 2.51225;
   DATA[542,1] := 534.2693;
   DATA[542,2] := 2.0;
   DATA[542,3] := 2.0;
   DATA[542,4] := 262.1764;
   DATA[542,5] := 8.395475;
   DATA[542,6] := 327.839;
   DATA[542,7] := 2.439753;
   DATA[542,8] := 2.0;
   DATA[542,9] := 2.0;
   DATA[542,10] := 2.0;
   DATA[542,11] := 19.72598;
   DATA[542,12] := 2.214265;
   DATA[542,13] := 980.8783;
   DATA[542,14] := 1.0;
   DATA[542,15] := 2.0;
   DATA[542,16] := 1.0;
   DATA[542,17] := 1.0;
   DATA[542,18] := 1.0;
   DATA[542,19] := 2.0;
   DATA[542,20] := 148.808;
   DATA[542,21] := 155.9344;
   DATA[542,22] := 1.72095;
   DATA[542,23] := 983.9016;
   DATA[542,24] := 2.0;
   DATA[542,25] := 2.0;
   DATA[542,26] := 7.87766;
   DATA[542,27] := 144.9628;
   DATA[542,28] := 263.4581;
   DATA[542,29] := 12.07383;
   DATA[542,30] := 1.730838;
   DATA[542,31] := 1.292686;
   DATA[542,32] := 0.7353967;
   DATA[542,33] := 0.3065689;
   DATA[542,34] := 2.0;
   DATA[542,35] := 251.0254;
   DATA[542,36] := 1.665972;
   DATA[542,37] := 189.759;
   DATA[542,38] := 0.000128152;
   DATA[542,39] := 1.0;
   DATA[543,0] := 2.500721;
   DATA[543,1] := 534.7403;
   DATA[543,2] := 2.0;
   DATA[543,3] := 2.0;
   DATA[543,4] := 262.1764;
   DATA[543,5] := 8.395475;
   DATA[543,6] := 327.839;
   DATA[543,7] := 2.439753;
   DATA[543,8] := 2.0;
   DATA[543,9] := 2.0;
   DATA[543,10] := 2.0;
   DATA[543,11] := 19.72598;
   DATA[543,12] := 2.2126;
   DATA[543,13] := 981.1587;
   DATA[543,14] := 1.0;
   DATA[543,15] := 2.0;
   DATA[543,16] := 1.0;
   DATA[543,17] := 1.0;
   DATA[543,18] := 1.0;
   DATA[543,19] := 2.0;
   DATA[543,20] := 148.808;
   DATA[543,21] := 155.9344;
   DATA[543,22] := 1.718002;
   DATA[543,23] := 984.5552;
   DATA[543,24] := 2.0;
   DATA[543,25] := 2.0;
   DATA[543,26] := 7.87766;
   DATA[543,27] := 144.6296;
   DATA[543,28] := 263.4581;
   DATA[543,29] := 12.07383;
   DATA[543,30] := 1.730838;
   DATA[543,31] := 1.292686;
   DATA[543,32] := 0.7353967;
   DATA[543,33] := 0.3065689;
   DATA[543,34] := 2.0;
   DATA[543,35] := 250.8972;
   DATA[543,36] := 1.665972;
   DATA[543,37] := 189.6469;
   DATA[543,38] := 0.000128152;
   DATA[543,39] := 1.0;
   DATA[544,0] := 2.481504;
   DATA[544,1] := 534.6226;
   DATA[544,2] := 2.0;
   DATA[544,3] := 2.0;
   DATA[544,4] := 262.1764;
   DATA[544,5] := 8.395475;
   DATA[544,6] := 327.839;
   DATA[544,7] := 2.441034;
   DATA[544,8] := 2.0;
   DATA[544,9] := 2.0;
   DATA[544,10] := 2.0;
   DATA[544,11] := 19.68756;
   DATA[544,12] := 2.212087;
   DATA[544,13] := 981.1587;
   DATA[544,14] := 1.0;
   DATA[544,15] := 2.0;
   DATA[544,16] := 1.0;
   DATA[544,17] := 1.0;
   DATA[544,18] := 1.0;
   DATA[544,19] := 2.0;
   DATA[544,20] := 148.808;
   DATA[544,21] := 155.9344;
   DATA[544,22] := 1.715824;
   DATA[544,23] := 984.9782;
   DATA[544,24] := 2.0;
   DATA[544,25] := 2.0;
   DATA[544,26] := 7.87766;
   DATA[544,27] := 144.6296;
   DATA[544,28] := 263.4581;
   DATA[544,29] := 12.07383;
   DATA[544,30] := 1.728531;
   DATA[544,31] := 1.292686;
   DATA[544,32] := 0.7353967;
   DATA[544,33] := 0.3065689;
   DATA[544,34] := 2.0;
   DATA[544,35] := 250.8972;
   DATA[544,36] := 1.665972;
   DATA[544,37] := 189.6469;
   DATA[544,38] := 0.000128152;
   DATA[544,39] := 1.0;
   DATA[545,0] := 2.458764;
   DATA[545,1] := 534.6226;
   DATA[545,2] := 2.0;
   DATA[545,3] := 2.0;
   DATA[545,4] := 262.1764;
   DATA[545,5] := 8.395475;
   DATA[545,6] := 327.839;
   DATA[545,7] := 2.442188;
   DATA[545,8] := 2.0;
   DATA[545,9] := 2.0;
   DATA[545,10] := 2.0;
   DATA[545,11] := 19.68436;
   DATA[545,12] := 2.210037;
   DATA[545,13] := 980.8783;
   DATA[545,14] := 1.0;
   DATA[545,15] := 2.0;
   DATA[545,16] := 1.0;
   DATA[545,17] := 1.0;
   DATA[545,18] := 1.0;
   DATA[545,19] := 2.0;
   DATA[545,20] := 148.808;
   DATA[545,21] := 155.9344;
   DATA[545,22] := 1.715824;
   DATA[545,23] := 985.4396;
   DATA[545,24] := 2.0;
   DATA[545,25] := 2.0;
   DATA[545,26] := 7.87766;
   DATA[545,27] := 144.6296;
   DATA[545,28] := 263.4581;
   DATA[545,29] := 12.07383;
   DATA[545,30] := 1.728531;
   DATA[545,31] := 1.292686;
   DATA[545,32] := 0.7353967;
   DATA[545,33] := 0.3065689;
   DATA[545,34] := 2.0;
   DATA[545,35] := 250.8972;
   DATA[545,36] := 1.665972;
   DATA[545,37] := 189.6469;
   DATA[545,38] := 0.000128152;
   DATA[545,39] := 1.0;
   DATA[546,0] := 2.447875;
   DATA[546,1] := 534.4263;
   DATA[546,2] := 2.0;
   DATA[546,3] := 2.0;
   DATA[546,4] := 262.1764;
   DATA[546,5] := 8.395475;
   DATA[546,6] := 327.839;
   DATA[546,7] := 2.442316;
   DATA[546,8] := 2.0;
   DATA[546,9] := 2.0;
   DATA[546,10] := 2.0;
   DATA[546,11] := 19.67155;
   DATA[546,12] := 2.209397;
   DATA[546,13] := 981.0385;
   DATA[546,14] := 1.0;
   DATA[546,15] := 2.0;
   DATA[546,16] := 1.0;
   DATA[546,17] := 1.0;
   DATA[546,18] := 1.0;
   DATA[546,19] := 2.0;
   DATA[546,20] := 148.808;
   DATA[546,21] := 155.9344;
   DATA[546,22] := 1.71467;
   DATA[546,23] := 985.9011;
   DATA[546,24] := 2.0;
   DATA[546,25] := 2.0;
   DATA[546,26] := 7.87766;
   DATA[546,27] := 144.6296;
   DATA[546,28] := 263.4581;
   DATA[546,29] := 12.07383;
   DATA[546,30] := 1.728531;
   DATA[546,31] := 1.275906;
   DATA[546,32] := 0.7353967;
   DATA[546,33] := 0.3065689;
   DATA[546,34] := 2.0;
   DATA[546,35] := 250.737;
   DATA[546,36] := 1.665972;
   DATA[546,37] := 189.6469;
   DATA[546,38] := 0.000128152;
   DATA[546,39] := 1.0;
   DATA[547,0] := 2.431861;
   DATA[547,1] := 533.7197;
   DATA[547,2] := 2.0;
   DATA[547,3] := 2.0;
   DATA[547,4] := 262.1764;
   DATA[547,5] := 8.395475;
   DATA[547,6] := 327.839;
   DATA[547,7] := 2.442316;
   DATA[547,8] := 2.0;
   DATA[547,9] := 2.0;
   DATA[547,10] := 2.0;
   DATA[547,11] := 19.61073;
   DATA[547,12] := 2.209397;
   DATA[547,13] := 980.8783;
   DATA[547,14] := 1.0;
   DATA[547,15] := 2.0;
   DATA[547,16] := 1.0;
   DATA[547,17] := 1.0;
   DATA[547,18] := 1.0;
   DATA[547,19] := 2.0;
   DATA[547,20] := 148.808;
   DATA[547,21] := 155.9344;
   DATA[547,22] := 1.713389;
   DATA[547,23] := 986.5547;
   DATA[547,24] := 2.0;
   DATA[547,25] := 2.0;
   DATA[547,26] := 7.87766;
   DATA[547,27] := 144.7578;
   DATA[547,28] := 263.4581;
   DATA[547,29] := 12.07383;
   DATA[547,30] := 1.728531;
   DATA[547,31] := 1.27898;
   DATA[547,32] := 0.7353967;
   DATA[547,33] := 0.3086186;
   DATA[547,34] := 2.0;
   DATA[547,35] := 250.721;
   DATA[547,36] := 1.665972;
   DATA[547,37] := 189.5668;
   DATA[547,38] := 0.000128152;
   DATA[547,39] := 1.0;
   DATA[548,0] := 2.422573;
   DATA[548,1] := 533.5627;
   DATA[548,2] := 2.0;
   DATA[548,3] := 2.0;
   DATA[548,4] := 262.1764;
   DATA[548,5] := 8.395475;
   DATA[548,6] := 327.839;
   DATA[548,7] := 2.442316;
   DATA[548,8] := 2.0;
   DATA[548,9] := 2.0;
   DATA[548,10] := 2.0;
   DATA[548,11] := 19.61073;
   DATA[548,12] := 2.209397;
   DATA[548,13] := 980.678;
   DATA[548,14] := 1.0;
   DATA[548,15] := 2.0;
   DATA[548,16] := 1.0;
   DATA[548,17] := 1.0;
   DATA[548,18] := 1.0;
   DATA[548,19] := 2.0;
   DATA[548,20] := 148.808;
   DATA[548,21] := 155.9344;
   DATA[548,22] := 1.713389;
   DATA[548,23] := 986.9777;
   DATA[548,24] := 2.0;
   DATA[548,25] := 2.0;
   DATA[548,26] := 7.87766;
   DATA[548,27] := 144.7578;
   DATA[548,28] := 263.4581;
   DATA[548,29] := 12.07383;
   DATA[548,30] := 1.726865;
   DATA[548,31] := 1.28103;
   DATA[548,32] := 0.7353967;
   DATA[548,33] := 0.3086186;
   DATA[548,34] := 2.0;
   DATA[548,35] := 250.721;
   DATA[548,36] := 1.665972;
   DATA[548,37] := 189.5668;
   DATA[548,38] := 0.000128152;
   DATA[548,39] := 1.0;
   DATA[549,0] := 2.417449;
   DATA[549,1] := 532.5814;
   DATA[549,2] := 2.0;
   DATA[549,3] := 2.0;
   DATA[549,4] := 262.1764;
   DATA[549,5] := 8.395475;
   DATA[549,6] := 327.839;
   DATA[549,7] := 2.442316;
   DATA[549,8] := 2.0;
   DATA[549,9] := 2.0;
   DATA[549,10] := 2.0;
   DATA[549,11] := 19.61073;
   DATA[549,12] := 2.205682;
   DATA[549,13] := 981.4791;
   DATA[549,14] := 1.0;
   DATA[549,15] := 2.0;
   DATA[549,16] := 1.0;
   DATA[549,17] := 1.0;
   DATA[549,18] := 1.0;
   DATA[549,19] := 2.0;
   DATA[549,20] := 148.808;
   DATA[549,21] := 155.9344;
   DATA[549,22] := 1.714029;
   DATA[549,23] := 987.7083;
   DATA[549,24] := 2.0;
   DATA[549,25] := 2.0;
   DATA[549,26] := 7.87766;
   DATA[549,27] := 144.7578;
   DATA[549,28] := 263.4581;
   DATA[549,29] := 12.07383;
   DATA[549,30] := 1.726865;
   DATA[549,31] := 1.285513;
   DATA[549,32] := 0.7353967;
   DATA[549,33] := 0.3075937;
   DATA[549,34] := 2.0;
   DATA[549,35] := 250.721;
   DATA[549,36] := 1.665972;
   DATA[549,37] := 189.5668;
   DATA[549,38] := 0.000128152;
   DATA[549,39] := 1.0;
   DATA[550,0] := 2.417449;
   DATA[550,1] := 532.5814;
   DATA[550,2] := 2.0;
   DATA[550,3] := 2.0;
   DATA[550,4] := 262.1764;
   DATA[550,5] := 8.395475;
   DATA[550,6] := 327.839;
   DATA[550,7] := 2.442316;
   DATA[550,8] := 2.0;
   DATA[550,9] := 2.0;
   DATA[550,10] := 2.0;
   DATA[550,11] := 19.61073;
   DATA[550,12] := 2.205682;
   DATA[550,13] := 981.4791;
   DATA[550,14] := 1.0;
   DATA[550,15] := 2.0;
   DATA[550,16] := 1.0;
   DATA[550,17] := 1.0;
   DATA[550,18] := 1.0;
   DATA[550,19] := 2.0;
   DATA[550,20] := 148.808;
   DATA[550,21] := 155.9344;
   DATA[550,22] := 1.714029;
   DATA[550,23] := 987.7083;
   DATA[550,24] := 2.0;
   DATA[550,25] := 2.0;
   DATA[550,26] := 7.87766;
   DATA[550,27] := 144.7578;
   DATA[550,28] := 263.4581;
   DATA[550,29] := 12.07383;
   DATA[550,30] := 1.726865;
   DATA[550,31] := 1.285513;
   DATA[550,32] := 0.7353967;
   DATA[550,33] := 0.3075937;
   DATA[550,34] := 2.0;
   DATA[550,35] := 250.721;
   DATA[550,36] := 1.665972;
   DATA[550,37] := 189.5668;
   DATA[550,38] := 0.000128152;
   DATA[550,39] := 1.0;
   DATA[551,0] := 2.423534;
   DATA[551,1] := 532.2674;
   DATA[551,2] := 2.0;
   DATA[551,3] := 2.0;
   DATA[551,4] := 262.1764;
   DATA[551,5] := 8.395475;
   DATA[551,6] := 327.839;
   DATA[551,7] := 2.441547;
   DATA[551,8] := 2.0;
   DATA[551,9] := 2.0;
   DATA[551,10] := 2.0;
   DATA[551,11] := 19.61073;
   DATA[551,12] := 2.205682;
   DATA[551,13] := 981.5593;
   DATA[551,14] := 1.0;
   DATA[551,15] := 2.0;
   DATA[551,16] := 1.0;
   DATA[551,17] := 1.0;
   DATA[551,18] := 1.0;
   DATA[551,19] := 2.0;
   DATA[551,20] := 148.808;
   DATA[551,21] := 155.9344;
   DATA[551,22] := 1.716849;
   DATA[551,23] := 988.0159;
   DATA[551,24] := 2.0;
   DATA[551,25] := 2.0;
   DATA[551,26] := 7.87766;
   DATA[551,27] := 144.7578;
   DATA[551,28] := 263.4581;
   DATA[551,29] := 12.07383;
   DATA[551,30] := 1.726865;
   DATA[551,31] := 1.291405;
   DATA[551,32] := 0.7353967;
   DATA[551,33] := 0.3065689;
   DATA[551,34] := 2.0;
   DATA[551,35] := 250.9773;
   DATA[551,36] := 1.665972;
   DATA[551,37] := 189.5668;
   DATA[551,38] := 0.000128152;
   DATA[551,39] := 1.0;
   DATA[552,0] := 2.455241;
   DATA[552,1] := 531.3253;
   DATA[552,2] := 2.0;
   DATA[552,3] := 2.0;
   DATA[552,4] := 262.1764;
   DATA[552,5] := 8.395475;
   DATA[552,6] := 327.839;
   DATA[552,7] := 2.441547;
   DATA[552,8] := 2.0;
   DATA[552,9] := 2.0;
   DATA[552,10] := 2.0;
   DATA[552,11] := 19.67155;
   DATA[552,12] := 2.208884;
   DATA[552,13] := 981.8796;
   DATA[552,14] := 1.0;
   DATA[552,15] := 2.0;
   DATA[552,16] := 1.0;
   DATA[552,17] := 1.0;
   DATA[552,18] := 1.0;
   DATA[552,19] := 2.0;
   DATA[552,20] := 148.808;
   DATA[552,21] := 155.9344;
   DATA[552,22] := 1.718771;
   DATA[552,23] := 987.939;
   DATA[552,24] := 2.0;
   DATA[552,25] := 2.0;
   DATA[552,26] := 7.87766;
   DATA[552,27] := 144.7578;
   DATA[552,28] := 263.4581;
   DATA[552,29] := 12.07383;
   DATA[552,30] := 1.726865;
   DATA[552,31] := 1.28436;
   DATA[552,32] := 0.7377012;
   DATA[552,33] := 0.3062486;
   DATA[552,34] := 2.0;
   DATA[552,35] := 251.0574;
   DATA[552,36] := 1.778105;
   DATA[552,37] := 189.743;
   DATA[552,38] := 0.000128152;
   DATA[552,39] := 1.0;
   DATA[553,0] := 2.494315;
   DATA[553,1] := 530.7758;
   DATA[553,2] := 2.0;
   DATA[553,3] := 2.0;
   DATA[553,4] := 262.1764;
   DATA[553,5] := 8.395475;
   DATA[553,6] := 327.839;
   DATA[553,7] := 2.441547;
   DATA[553,8] := 2.0;
   DATA[553,9] := 2.0;
   DATA[553,10] := 2.0;
   DATA[553,11] := 19.70037;
   DATA[553,12] := 2.208884;
   DATA[553,13] := 981.7595;
   DATA[553,14] := 1.0;
   DATA[553,15] := 2.0;
   DATA[553,16] := 1.0;
   DATA[553,17] := 1.0;
   DATA[553,18] := 1.0;
   DATA[553,19] := 2.0;
   DATA[553,20] := 148.808;
   DATA[553,21] := 155.9344;
   DATA[553,22] := 1.719924;
   DATA[553,23] := 988.2081;
   DATA[553,24] := 2.0;
   DATA[553,25] := 2.0;
   DATA[553,26] := 7.878942;
   DATA[553,27] := 144.7578;
   DATA[553,28] := 263.4581;
   DATA[553,29] := 12.07383;
   DATA[553,30] := 1.726865;
   DATA[553,31] := 1.281542;
   DATA[553,32] := 0.7377012;
   DATA[553,33] := 0.3062486;
   DATA[553,34] := 2.0;
   DATA[553,35] := 251.2016;
   DATA[553,36] := 1.778105;
   DATA[553,37] := 189.8231;
   DATA[553,38] := 0.000128152;
   DATA[553,39] := 1.0;
   DATA[554,0] := 2.54652;
   DATA[554,1] := 529.7159;
   DATA[554,2] := 2.0;
   DATA[554,3] := 2.0;
   DATA[554,4] := 262.1764;
   DATA[554,5] := 8.395475;
   DATA[554,6] := 327.839;
   DATA[554,7] := 2.441547;
   DATA[554,8] := 2.0;
   DATA[554,9] := 2.0;
   DATA[554,10] := 2.0;
   DATA[554,11] := 19.71637;
   DATA[554,12] := 2.208884;
   DATA[554,13] := 981.5593;
   DATA[554,14] := 1.0;
   DATA[554,15] := 2.0;
   DATA[554,16] := 1.0;
   DATA[554,17] := 1.0;
   DATA[554,18] := 1.0;
   DATA[554,19] := 2.0;
   DATA[554,20] := 148.808;
   DATA[554,21] := 155.9344;
   DATA[554,22] := 1.723256;
   DATA[554,23] := 988.5157;
   DATA[554,24] := 2.0;
   DATA[554,25] := 2.0;
   DATA[554,26] := 7.880544;
   DATA[554,27] := 144.7578;
   DATA[554,28] := 263.4581;
   DATA[554,29] := 12.07383;
   DATA[554,30] := 1.726865;
   DATA[554,31] := 1.281542;
   DATA[554,32] := 0.7377012;
   DATA[554,33] := 0.3062486;
   DATA[554,34] := 2.0;
   DATA[554,35] := 251.2977;
   DATA[554,36] := 1.778105;
   DATA[554,37] := 189.9833;
   DATA[554,38] := 0.000128152;
   DATA[554,39] := 1.0;
   DATA[555,0] := 2.570541;
   DATA[555,1] := 529.3627;
   DATA[555,2] := 2.0;
   DATA[555,3] := 2.0;
   DATA[555,4] := 262.1764;
   DATA[555,5] := 8.395475;
   DATA[555,6] := 327.839;
   DATA[555,7] := 2.441547;
   DATA[555,8] := 2.0;
   DATA[555,9] := 2.0;
   DATA[555,10] := 2.0;
   DATA[555,11] := 19.75159;
   DATA[555,12] := 2.208884;
   DATA[555,13] := 981.2789;
   DATA[555,14] := 1.0;
   DATA[555,15] := 2.0;
   DATA[555,16] := 1.0;
   DATA[555,17] := 1.0;
   DATA[555,18] := 1.0;
   DATA[555,19] := 2.0;
   DATA[555,20] := 148.808;
   DATA[555,21] := 155.9344;
   DATA[555,22] := 1.724153;
   DATA[555,23] := 988.4388;
   DATA[555,24] := 2.0;
   DATA[555,25] := 2.0;
   DATA[555,26] := 7.880544;
   DATA[555,27] := 144.7578;
   DATA[555,28] := 263.4581;
   DATA[555,29] := 12.07383;
   DATA[555,30] := 1.728019;
   DATA[555,31] := 1.288715;
   DATA[555,32] := 0.7379573;
   DATA[555,33] := 0.3062486;
   DATA[555,34] := 2.0;
   DATA[555,35] := 251.2977;
   DATA[555,36] := 1.778105;
   DATA[555,37] := 190.0474;
   DATA[555,38] := 0.000128152;
   DATA[555,39] := 1.0;
   DATA[556,0] := 2.61634;
   DATA[556,1] := 528.5776;
   DATA[556,2] := 2.0;
   DATA[556,3] := 2.0;
   DATA[556,4] := 262.1764;
   DATA[556,5] := 8.395475;
   DATA[556,6] := 327.839;
   DATA[556,7] := 2.441547;
   DATA[556,8] := 2.0;
   DATA[556,9] := 2.0;
   DATA[556,10] := 2.0;
   DATA[556,11] := 19.79;
   DATA[556,12] := 2.208372;
   DATA[556,13] := 981.1987;
   DATA[556,14] := 1.0;
   DATA[556,15] := 2.0;
   DATA[556,16] := 1.0;
   DATA[556,17] := 1.0;
   DATA[556,18] := 1.0;
   DATA[556,19] := 2.0;
   DATA[556,20] := 148.808;
   DATA[556,21] := 156.0369;
   DATA[556,22] := 1.724153;
   DATA[556,23] := 989.0156;
   DATA[556,24] := 2.0;
   DATA[556,25] := 2.0;
   DATA[556,26] := 7.880544;
   DATA[556,27] := 144.7578;
   DATA[556,28] := 263.4581;
   DATA[556,29] := 12.07383;
   DATA[556,30] := 1.729172;
   DATA[556,31] := 1.292558;
   DATA[556,32] := 0.7357808;
   DATA[556,33] := 0.3066329;
   DATA[556,34] := 2.0;
   DATA[556,35] := 251.2977;
   DATA[556,36] := 1.778105;
   DATA[556,37] := 190.0474;
   DATA[556,38] := 0.000128152;
   DATA[556,39] := 1.0;
   DATA[557,0] := 2.641322;
   DATA[557,1] := 528.4599;
   DATA[557,2] := 2.0;
   DATA[557,3] := 2.0;
   DATA[557,4] := 262.1764;
   DATA[557,5] := 8.395475;
   DATA[557,6] := 327.9159;
   DATA[557,7] := 2.441162;
   DATA[557,8] := 2.0;
   DATA[557,9] := 2.0;
   DATA[557,10] := 2.0;
   DATA[557,11] := 19.80601;
   DATA[557,12] := 2.208372;
   DATA[557,13] := 981.4391;
   DATA[557,14] := 1.0;
   DATA[557,15] := 2.0;
   DATA[557,16] := 1.0;
   DATA[557,17] := 1.0;
   DATA[557,18] := 1.0;
   DATA[557,19] := 2.0;
   DATA[557,20] := 148.808;
   DATA[557,21] := 156.0369;
   DATA[557,22] := 1.724153;
   DATA[557,23] := 988.708;
   DATA[557,24] := 2.0;
   DATA[557,25] := 2.0;
   DATA[557,26] := 7.880544;
   DATA[557,27] := 144.7578;
   DATA[557,28] := 263.4581;
   DATA[557,29] := 12.07383;
   DATA[557,30] := 1.729172;
   DATA[557,31] := 1.292558;
   DATA[557,32] := 0.7357808;
   DATA[557,33] := 0.3066329;
   DATA[557,34] := 2.0;
   DATA[557,35] := 251.2977;
   DATA[557,36] := 1.778105;
   DATA[557,37] := 190.0474;
   DATA[557,38] := 0.000128152;
   DATA[557,39] := 1.0;
   DATA[558,0] := 2.672389;
   DATA[558,1] := 528.8132;
   DATA[558,2] := 2.0;
   DATA[558,3] := 2.0;
   DATA[558,4] := 262.1764;
   DATA[558,5] := 8.395475;
   DATA[558,6] := 327.9159;
   DATA[558,7] := 2.440265;
   DATA[558,8] := 2.0;
   DATA[558,9] := 2.0;
   DATA[558,10] := 2.0;
   DATA[558,11] := 19.80601;
   DATA[558,12] := 2.210806;
   DATA[558,13] := 981.7996;
   DATA[558,14] := 1.0;
   DATA[558,15] := 2.0;
   DATA[558,16] := 1.0;
   DATA[558,17] := 1.0;
   DATA[558,18] := 1.0;
   DATA[558,19] := 2.0;
   DATA[558,20] := 148.808;
   DATA[558,21] := 156.0369;
   DATA[558,22] := 1.724153;
   DATA[558,23] := 988.9003;
   DATA[558,24] := 2.0;
   DATA[558,25] := 2.0;
   DATA[558,26] := 7.880544;
   DATA[558,27] := 144.7578;
   DATA[558,28] := 263.4581;
   DATA[558,29] := 12.07383;
   DATA[558,30] := 1.729172;
   DATA[558,31] := 1.292174;
   DATA[558,32] := 0.7357808;
   DATA[558,33] := 0.3074656;
   DATA[558,34] := 2.0;
   DATA[558,35] := 251.2977;
   DATA[558,36] := 1.778105;
   DATA[558,37] := 190.0474;
   DATA[558,38] := 0.000128152;
   DATA[558,39] := 1.0;
   DATA[559,0] := 2.674951;
   DATA[559,1] := 528.7739;
   DATA[559,2] := 2.0;
   DATA[559,3] := 2.0;
   DATA[559,4] := 262.1764;
   DATA[559,5] := 8.395475;
   DATA[559,6] := 327.9159;
   DATA[559,7] := 2.440265;
   DATA[559,8] := 2.0;
   DATA[559,9] := 2.0;
   DATA[559,10] := 2.0;
   DATA[559,11] := 19.73238;
   DATA[559,12] := 2.211959;
   DATA[559,13] := 981.5993;
   DATA[559,14] := 1.0;
   DATA[559,15] := 2.0;
   DATA[559,16] := 1.0;
   DATA[559,17] := 1.0;
   DATA[559,18] := 1.0;
   DATA[559,19] := 2.0;
   DATA[559,20] := 148.808;
   DATA[559,21] := 156.0369;
   DATA[559,22] := 1.723641;
   DATA[559,23] := 988.6696;
   DATA[559,24] := 2.0;
   DATA[559,25] := 2.0;
   DATA[559,26] := 7.880544;
   DATA[559,27] := 144.7578;
   DATA[559,28] := 263.4581;
   DATA[559,29] := 12.07383;
   DATA[559,30] := 1.730838;
   DATA[559,31] := 1.283079;
   DATA[559,32] := 0.7353967;
   DATA[559,33] := 0.3080421;
   DATA[559,34] := 2.0;
   DATA[559,35] := 251.2977;
   DATA[559,36] := 1.746067;
   DATA[559,37] := 190.0474;
   DATA[559,38] := 0.000128152;
   DATA[559,39] := 1.0;
   DATA[560,0] := 2.643244;
   DATA[560,1] := 529.6375;
   DATA[560,2] := 2.0;
   DATA[560,3] := 2.0;
   DATA[560,4] := 262.1764;
   DATA[560,5] := 8.395475;
   DATA[560,6] := 327.9159;
   DATA[560,7] := 2.4427;
   DATA[560,8] := 2.0;
   DATA[560,9] := 2.0;
   DATA[560,10] := 2.0;
   DATA[560,11] := 19.69076;
   DATA[560,12] := 2.211959;
   DATA[560,13] := 981.1987;
   DATA[560,14] := 1.0;
   DATA[560,15] := 2.0;
   DATA[560,16] := 1.0;
   DATA[560,17] := 1.0;
   DATA[560,18] := 1.0;
